       #MyWord := "EPICSToPLC"."Word"[#EPICSToPLCDataBlockOffset + 0];
       "EPICSToPLC"."Word"[#EPICSToPLCDataBlockOffset + 0] := 0;
       #"Cmd_Stop_system" := #MyBoolsinWord[8];    //EPICSName: Cmd_Stop_system
       #"Cmd_Start_system" := #MyBoolsinWord[9];    //EPICSName: Cmd_Start_system
       #"Cmd_Stand_by_4K" := #MyBoolsinWord[10];    //EPICSName: Cmd_Stand_by_4K
       #"Cmd_Stand_by_2K" := #MyBoolsinWord[11];    //EPICSName: Cmd_Stand_by_2K
       #"Cmd_Nominal_2K_RF" := #MyBoolsinWord[12];    //EPICSName: Cmd_Nominal_2K_RF
       #"Cmd_Stand_by_300K" := #MyBoolsinWord[13];    //EPICSName: Cmd_Stand_by_300K
       #"Cmd_Stand_by_80K" := #MyBoolsinWord[14];    //EPICSName: Cmd_Stand_by_80K
       #"Cmd_Reset" := #MyBoolsinWord[15];    //EPICSName: Cmd_Reset
    Else
       #DEVICE_PARAM_OK := FALSE; //Invalid Hash
    END_IF;
END_FUNCTION_BLOCK
FUNCTION_BLOCK "DEVTYPE_C3S_PID"
{ S7_Optimized_Access := 'TRUE' }
VERSION : 1.0
   VAR_INPUT
      "OpMode_Auto" { ExternalAccessible := 'True'; ExternalVisible := 'False'; ExternalWritable := 'False'; } : BOOL;   //EPICS Status variable: OpMode_Auto
      "OpMode_Manual" { ExternalAccessible := 'True'; ExternalVisible := 'False'; ExternalWritable := 'False'; } : BOOL;   //EPICS Status variable: OpMode_Manual
      "OpMode_Forced" { ExternalAccessible := 'True'; ExternalVisible := 'False'; ExternalWritable := 'False'; } : BOOL;   //EPICS Status variable: OpMode_Forced
      "PID_Color" { ExternalAccessible := 'True'; ExternalVisible := 'False'; ExternalWritable := 'False'; } : INT;   //EPICS Status variable: PID_Color
      "LMN" { ExternalAccessible := 'True'; ExternalVisible := 'False'; ExternalWritable := 'False'; } : REAL;   //EPICS Status variable: LMN
      "LMN_P" { ExternalAccessible := 'True'; ExternalVisible := 'False'; ExternalWritable := 'False'; } : REAL;   //EPICS Status variable: LMN_P
      "LMN_I" { ExternalAccessible := 'True'; ExternalVisible := 'False'; ExternalWritable := 'False'; } : REAL;   //EPICS Status variable: LMN_I
      "LMN_D" { ExternalAccessible := 'True'; ExternalVisible := 'False'; ExternalWritable := 'False'; } : REAL;   //EPICS Status variable: LMN_D
      "PID_DIF" { ExternalAccessible := 'True'; ExternalVisible := 'False'; ExternalWritable := 'False'; } : REAL;   //EPICS Status variable: PID_DIF
      "PV" { ExternalAccessible := 'True'; ExternalVisible := 'False'; ExternalWritable := 'False'; } : REAL;   //EPICS Status variable: PV
      "MAN_SP" { ExternalAccessible := 'True'; ExternalVisible := 'False'; ExternalWritable := 'False'; } : REAL;   //EPICS Status variable: MAN_SP
      "PID_Cycle" { ExternalAccessible := 'True'; ExternalVisible := 'False'; ExternalWritable := 'False'; } : INT;   //EPICS Status variable: PID_Cycle
      "ProcValueName" { ExternalAccessible := 'True'; ExternalVisible := 'False'; ExternalWritable := 'False'; } : STRING;   //EPICS Status variable: ProcValueName
      "ProcValueEGU" { ExternalAccessible := 'True'; ExternalVisible := 'False'; ExternalWritable := 'False'; } : STRING;   //EPICS Status variable: ProcValueEGU
      "Inhibit_Manual" { ExternalAccessible := 'True'; ExternalVisible := 'False'; ExternalWritable := 'False'; } : BOOL;   //EPICS Status variable: Inhibit_Manual
      "Inhibit_Force" { ExternalAccessible := 'True'; ExternalVisible := 'False'; ExternalWritable := 'False'; } : BOOL;   //EPICS Status variable: Inhibit_Force
      "Inhibit_Lock" { ExternalAccessible := 'True'; ExternalVisible := 'False'; ExternalWritable := 'False'; } : BOOL;   //EPICS Status variable: Inhibit_Lock
      "MoveInterlock" { ExternalAccessible := 'True'; ExternalVisible := 'False'; ExternalWritable := 'False'; } : BOOL;   //EPICS Status variable: MoveInterlock
      "GroupInterlock" { ExternalAccessible := 'True'; ExternalVisible := 'False'; ExternalWritable := 'False'; } : BOOL;   //EPICS Status variable: GroupInterlock
      "EnableAutoBtn" { ExternalAccessible := 'True'; ExternalVisible := 'False'; ExternalWritable := 'False'; } : BOOL;   //EPICS Status variable: EnableAutoBtn
      "EnableManualBtn" { ExternalAccessible := 'True'; ExternalVisible := 'False'; ExternalWritable := 'False'; } : BOOL;   //EPICS Status variable: EnableManualBtn
      "EnableForcedBtn" { ExternalAccessible := 'True'; ExternalVisible := 'False'; ExternalWritable := 'False'; } : BOOL;   //EPICS Status variable: EnableForcedBtn
      "EnablePIDConf" { ExternalAccessible := 'True'; ExternalVisible := 'False'; ExternalWritable := 'False'; } : BOOL;   //EPICS Status variable: EnablePIDConf
      "LatchAlarm" { ExternalAccessible := 'True'; ExternalVisible := 'False'; ExternalWritable := 'False'; } : BOOL;   //EPICS Status variable: LatchAlarm
      "GroupAlarm" { ExternalAccessible := 'True'; ExternalVisible := 'False'; ExternalWritable := 'False'; } : BOOL;   //EPICS Status variable: GroupAlarm
      "EnableBlkCtrl" { ExternalAccessible := 'True'; ExternalVisible := 'False'; ExternalWritable := 'False'; } : BOOL;   //EPICS Status variable: EnableBlkCtrl
      "EnableForceValBtn" { ExternalAccessible := 'True'; ExternalVisible := 'False'; ExternalWritable := 'False'; } : BOOL;   //EPICS Status variable: EnableForceValBtn
      "DevLocked" { ExternalAccessible := 'True'; ExternalVisible := 'False'; ExternalWritable := 'False'; } : BOOL;   //EPICS Status variable: DevLocked
      "Faceplate_LockID" { ExternalAccessible := 'True'; ExternalVisible := 'False'; ExternalWritable := 'False'; } : DINT;   //EPICS Status variable: Faceplate_LockID
      "BlockIcon_LockID" { ExternalAccessible := 'True'; ExternalVisible := 'False'; ExternalWritable := 'False'; } : DINT;   //EPICS Status variable: BlockIcon_LockID
      "LMN_HLIM" { ExternalAccessible := 'True'; ExternalVisible := 'False'; ExternalWritable := 'False'; } : BOOL;   //EPICS Status variable: LMN_HLIM
      "LMN_LLIM" { ExternalAccessible := 'True'; ExternalVisible := 'False'; ExternalWritable := 'False'; } : BOOL;   //EPICS Status variable: LMN_LLIM
      "IO_Error" { ExternalAccessible := 'True'; ExternalVisible := 'False'; ExternalWritable := 'False'; } : BOOL;   //EPICS Status variable: IO_Error
      "Input_Module_Error" { ExternalAccessible := 'True'; ExternalVisible := 'False'; ExternalWritable := 'False'; } : BOOL;   //EPICS Status variable: Input_Module_Error
      "Output_Module_Error" { ExternalAccessible := 'True'; ExternalVisible := 'False'; ExternalWritable := 'False'; } : BOOL;   //EPICS Status variable: Output_Module_Error
      "Discrepancy_Error" { ExternalAccessible := 'True'; ExternalVisible := 'False'; ExternalWritable := 'False'; } : BOOL;   //EPICS Status variable: Discrepancy_Error
      "ContDeviceInMan" { ExternalAccessible := 'True'; ExternalVisible := 'False'; ExternalWritable := 'False'; } : BOOL;   //EPICS Status variable: ContDeviceInMan
      "FB_Gain" { ExternalAccessible := 'True'; ExternalVisible := 'False'; ExternalWritable := 'False'; } : REAL;   //EPICS Status variable: FB_Gain
      "FB_TI" { ExternalAccessible := 'True'; ExternalVisible := 'False'; ExternalWritable := 'False'; } : DINT;   //EPICS Status variable: FB_TI
      "FB_TD" { ExternalAccessible := 'True'; ExternalVisible := 'False'; ExternalWritable := 'False'; } : DINT;   //EPICS Status variable: FB_TD
      "FB_DEADB" { ExternalAccessible := 'True'; ExternalVisible := 'False'; ExternalWritable := 'False'; } : REAL;   //EPICS Status variable: FB_DEADB
      "FB_LMN_HLIM" { ExternalAccessible := 'True'; ExternalVisible := 'False'; ExternalWritable := 'False'; } : REAL;   //EPICS Status variable: FB_LMN_HLIM
      "FB_LMN_LLIM" { ExternalAccessible := 'True'; ExternalVisible := 'False'; ExternalWritable := 'False'; } : REAL;   //EPICS Status variable: FB_LMN_LLIM
      "FB_ForcePosition" { ExternalAccessible := 'True'; ExternalVisible := 'False'; ExternalWritable := 'False'; } : REAL;   //EPICS Status variable: FB_ForcePosition
      "FB_Setpoint" { ExternalAccessible := 'True'; ExternalVisible := 'False'; ExternalWritable := 'False'; } : REAL;   //EPICS Status variable: FB_Setpoint
      "FB_Step" { ExternalAccessible := 'True'; ExternalVisible := 'False'; ExternalWritable := 'False'; } : REAL;   //EPICS Status variable: FB_Step
      "FB_Manipulated" { ExternalAccessible := 'True'; ExternalVisible := 'False'; ExternalWritable := 'False'; } : REAL;   //EPICS Status variable: FB_Manipulated
      "FB_P_ActionState" { ExternalAccessible := 'True'; ExternalVisible := 'False'; ExternalWritable := 'False'; } : BOOL;   //EPICS Status variable: FB_P_ActionState
      "FB_I_ActionState" { ExternalAccessible := 'True'; ExternalVisible := 'False'; ExternalWritable := 'False'; } : BOOL;   //EPICS Status variable: FB_I_ActionState
      "FB_D_ActionState" { ExternalAccessible := 'True'; ExternalVisible := 'False'; ExternalWritable := 'False'; } : BOOL;   //EPICS Status variable: FB_D_ActionState
      "FB_SS_State" { ExternalAccessible := 'True'; ExternalVisible := 'False'; ExternalWritable := 'False'; } : BOOL;   //EPICS Status variable: FB_SS_State
      "FB_SS_Value" { ExternalAccessible := 'True'; ExternalVisible := 'False'; ExternalWritable := 'False'; } : REAL;   //EPICS Status variable: FB_SS_Value
      "MeasValue_Msg" { ExternalAccessible := 'True'; ExternalVisible := 'False'; ExternalWritable := 'False'; } : STRING;   //EPICS Status variable: Measured_Value_Msg
   EPICSToPLCLength { ExternalAccessible := 'False'; ExternalVisible := 'False'; ExternalWritable := 'False'; } : Int;   // Length of device command register array (in words)
   EPICSToPLCDataBlockOffset { ExternalAccessible := 'False'; ExternalVisible := 'False'; ExternalWritable := 'False'; } : Int;   // Offset in EPICS->PLC comms block where this device data resides (in words)
   PLCToEPICSLength { ExternalAccessible := 'False'; ExternalVisible := 'False'; ExternalWritable := 'False'; } : Int;   // Length of device status register array (in words)
   PLCToEPICSDataBlockOffset { ExternalAccessible := 'False'; ExternalVisible := 'False'; ExternalWritable := 'False'; } : Int;   // Offset in PLC->EPICS comms block where this device data resides (in words)
   END_VAR
   VAR_OUTPUT
      "Cmd_Auto" { ExternalAccessible := 'True'; ExternalVisible := 'False'; ExternalWritable := 'False'; } : BOOL;   //EPICS Command variable: Cmd_Auto
      "Cmd_Manual" { ExternalAccessible := 'True'; ExternalVisible := 'False'; ExternalWritable := 'False'; } : BOOL;   //EPICS Command variable: Cmd_Manual
      "Cmd_Force" { ExternalAccessible := 'True'; ExternalVisible := 'False'; ExternalWritable := 'False'; } : BOOL;   //EPICS Command variable: Cmd_Force
      "Cmd_EnablePID_Conf" { ExternalAccessible := 'True'; ExternalVisible := 'False'; ExternalWritable := 'False'; } : BOOL;   //EPICS Command variable: Cmd_EnablePID_Conf
      "Cmd_DisablePID_Conf" { ExternalAccessible := 'True'; ExternalVisible := 'False'; ExternalWritable := 'False'; } : BOOL;   //EPICS Command variable: Cmd_DisablePID_Conf
      "Cmd_P_ON" { ExternalAccessible := 'True'; ExternalVisible := 'False'; ExternalWritable := 'False'; } : BOOL;   //EPICS Command variable: Cmd_P_ON
      "Cmd_P_OFF" { ExternalAccessible := 'True'; ExternalVisible := 'False'; ExternalWritable := 'False'; } : BOOL;   //EPICS Command variable: Cmd_P_OFF
      "Cmd_I_ON" { ExternalAccessible := 'True'; ExternalVisible := 'False'; ExternalWritable := 'False'; } : BOOL;   //EPICS Command variable: Cmd_I_ON
      "Cmd_I_OFF" { ExternalAccessible := 'True'; ExternalVisible := 'False'; ExternalWritable := 'False'; } : BOOL;   //EPICS Command variable: Cmd_I_OFF
      "Cmd_D_ON" { ExternalAccessible := 'True'; ExternalVisible := 'False'; ExternalWritable := 'False'; } : BOOL;   //EPICS Command variable: Cmd_D_ON
      "Cmd_D_OFF" { ExternalAccessible := 'True'; ExternalVisible := 'False'; ExternalWritable := 'False'; } : BOOL;   //EPICS Command variable: Cmd_D_OFF
      "Cmd_AckAlarm" { ExternalAccessible := 'True'; ExternalVisible := 'False'; ExternalWritable := 'False'; } : BOOL;   //EPICS Command variable: Cmd_AckAlarm
      "Cmd_ForceValInp" { ExternalAccessible := 'True'; ExternalVisible := 'False'; ExternalWritable := 'False'; } : BOOL;   //EPICS Command variable: Cmd_ForceValInp
      "Cmd_ForceValOut" { ExternalAccessible := 'True'; ExternalVisible := 'False'; ExternalWritable := 'False'; } : BOOL;   //EPICS Command variable: Cmd_ForceValOut
      "Cmd_ForceUnlock" { ExternalAccessible := 'True'; ExternalVisible := 'False'; ExternalWritable := 'False'; } : BOOL;   //EPICS Command variable: Cmd_ForceUnlock
      "Cmd_DevLock" { ExternalAccessible := 'True'; ExternalVisible := 'False'; ExternalWritable := 'False'; } : BOOL;   //EPICS Command variable: Cmd_DevLock
      "Cmd_DevUnlock" { ExternalAccessible := 'True'; ExternalVisible := 'False'; ExternalWritable := 'False'; } : BOOL;   //EPICS Command variable: Cmd_DevUnlock
      "P_Gain" { ExternalAccessible := 'True'; ExternalVisible := 'False'; ExternalWritable := 'False'; } : REAL;   //EPICS Parameter variable: P_Gain
      "P_TI" { ExternalAccessible := 'True'; ExternalVisible := 'False'; ExternalWritable := 'False'; } : DINT;   //EPICS Parameter variable: P_TI
      "P_TD" { ExternalAccessible := 'True'; ExternalVisible := 'False'; ExternalWritable := 'False'; } : DINT;   //EPICS Parameter variable: P_TD
      "P_DEADB" { ExternalAccessible := 'True'; ExternalVisible := 'False'; ExternalWritable := 'False'; } : REAL;   //EPICS Parameter variable: P_DEADB
      "P_LMN_HLIM" { ExternalAccessible := 'True'; ExternalVisible := 'False'; ExternalWritable := 'False'; } : REAL;   //EPICS Parameter variable: P_LMN_HLIM
      "P_LMN_LLIM" { ExternalAccessible := 'True'; ExternalVisible := 'False'; ExternalWritable := 'False'; } : REAL;   //EPICS Parameter variable: P_LMN_LLIM
      "P_ForcePosition" { ExternalAccessible := 'True'; ExternalVisible := 'False'; ExternalWritable := 'False'; } : REAL;   //EPICS Parameter variable: P_ForcePosition
      "P_Setpoint" { ExternalAccessible := 'True'; ExternalVisible := 'False'; ExternalWritable := 'False'; } : REAL;   //EPICS Parameter variable: P_Setpoint
      "P_Manipulated" { ExternalAccessible := 'True'; ExternalVisible := 'False'; ExternalWritable := 'False'; } : REAL;   //EPICS Parameter variable: P_Manipulated
      "P_Step" { ExternalAccessible := 'True'; ExternalVisible := 'False'; ExternalWritable := 'False'; } : REAL;   //EPICS Parameter variable: P_Step
      "P_Faceplate_LockID" { ExternalAccessible := 'True'; ExternalVisible := 'False'; ExternalWritable := 'False'; } : DINT;   //EPICS Parameter variable: P_Faceplate_LockID
      "P_BlockIcon_LockID" { ExternalAccessible := 'True'; ExternalVisible := 'False'; ExternalWritable := 'False'; } : DINT;   //EPICS Parameter variable: P_BlockIcon_LockID
      DEVICE_PARAM_OK { ExternalAccessible := 'False'; ExternalVisible := 'False'; ExternalWritable := 'False'; } : Bool;
   END_VAR
   VAR_IN_OUT
   END_VAR
   Var DB_SPECIFIC
      MyWord { ExternalAccessible := 'False'; ExternalVisible := 'False'; ExternalWritable := 'False'; } : Word;
      MyBytesinWord { ExternalAccessible := 'False'; ExternalVisible := 'False'; ExternalWritable := 'False'; } AT MyWord : Array[0..1] of Byte;
      MyBoolsinWord { ExternalAccessible := 'False'; ExternalVisible := 'False'; ExternalWritable := 'False'; } AT MyWord : Array[0..15] of Bool;
      MyDInt { ExternalAccessible := 'False'; ExternalVisible := 'False'; ExternalWritable := 'False'; } : DInt;
      MyWordsinDint { ExternalAccessible := 'False'; ExternalVisible := 'False'; ExternalWritable := 'False'; } AT MyDInt : Array[0..1] of Word;
      MyReal { ExternalAccessible := 'False'; ExternalVisible := 'False'; ExternalWritable := 'False'; } : Real;
      MyWordsinReal { ExternalAccessible := 'False'; ExternalVisible := 'False'; ExternalWritable := 'False'; } AT MyReal : Array[0..1] of Word;
      MyInt { ExternalAccessible := 'False'; ExternalVisible := 'False'; ExternalWritable := 'False'; } : Int;
      MyWordinInt { ExternalAccessible := 'False'; ExternalVisible := 'False'; ExternalWritable := 'False'; } AT MyInt : Word;
      MyDWord { ExternalAccessible := 'False'; ExternalVisible := 'False'; ExternalWritable := 'False'; } : DWord;
      MyWordsinDWord { ExternalAccessible := 'False'; ExternalVisible := 'False'; ExternalWritable := 'False'; } AT MyDWord : Array[0..1] of Word;
      MyTime { ExternalAccessible := 'False'; ExternalVisible := 'False'; ExternalWritable := 'False'; } : Time;
      MyWordsinTime { ExternalAccessible := 'False'; ExternalVisible := 'False'; ExternalWritable := 'False'; } AT MyTime : Array[0..1] of Word;
      MyString { ExternalAccessible := 'False'; ExternalVisible := 'False'; ExternalWritable := 'False'; } : String[40];
      MyWordsinString { ExternalAccessible := 'False'; ExternalVisible := 'False'; ExternalWritable := 'False'; } AT MyString : Array[0..20] of Word;
   END_VAR
   VAR_TEMP
      HashModbus : DInt;
      HashIFA : DInt;
      HashTIAMap : DInt;
      i : Int;
   END_VAR
    //Author: Miklos Boros (miklos.boros@esss.se), Copyrigth 2017-2020 by European Spallation Source, Lund
    //This block was generated by PLCFactory, please don't change it MANUALLY!
    //Input File Name: Spk-000CDL_Cryo-PLC-010-template-IFA-20220922093722.ifa
    //Generated: 20220922093722
    //According to HASH: 457744924
    //Device type: C3S_PID
    //Description: This function does the variable mapping for a device. All device-variable will be linked to an interface variable defined in this block.

    //********************************************
    //****************HASH check******************
    //********************************************


    #MyWordsinDint[0] := "EPICSToPLC"."Word"[0];
    #MyWordsinDint[1] := "EPICSToPLC"."Word"[1];
    #HashModbus := #MyDInt; //Hash from EPICS/ModbusTCP

    #HashIFA := 457744924; //Hash from Interface Factory as a constant

    #MyWordsinDint[0] := "PLCToEPICS"."Word"[0];
    #MyWordsinDint[1] := "PLCToEPICS"."Word"[1];
    #HashTIAMap := #MyDInt; //Hash from PLCFactory TIA Map


    IF ((#HashIFA = #HashModbus) AND (#HashModbus = #HashTIAMap)) THEN //Check CRCs
        #DEVICE_PARAM_OK := TRUE;
       //##################################### ICS HWI ###############################################
       //############################  ICS Instrument Library     ####################################
       //#  PLC Sample Code in VersionDog: ICS_LIBRARY_MASTER_PLC                                   ##
       //#  CCDB device types: ICS_xxxxx                                                            ##
       //#  EPICS HMI (Block Icons/Faceplates)@ GitLab. Projekt: Cryo / CryogenicsLibrary / CryoLib ##
       //#                                                                                          ##
       //#                                 PID - PID Control                                        ##
       //#                                                                                          ##
       //#                                                                                          ##
       //###########################           Version: 1.2           ################################
       //Author:	Zoltan Madi
       //Date:		13-12-2019
       //Version:  v1.2
       //Changes:  Added "MeasValue_Msg"
       //###########################           Version: 1.1           ################################
       //Author:	Johannes Kazantzidis
       //Date:		13-12-2019
       //Version:  v1.1
       //Changes:  Added alarm signal "Discrepancy_Error"
       //###########################           Version: 1.0           ################################
       //Author:	Miklos Boros
       //Date:		01-09-2019
       //Version:  v1.0
       //Changes:  First release and alarm signal "Discrepancy_Error"
       //#############################################################################################
       //###########################
       //STATUS BLOCK
       //###########################
       //Operation modes
       //OPI buttons
       //PID

    //********************************************
    //*************STATUS VARIABLES***************
    //********************************************


       #MyWord := W#0;
       #MyBoolsinWord[8] := #"OpMode_Auto";    //EPICSName: OpMode_Auto
       #MyBoolsinWord[9] := #"OpMode_Manual";    //EPICSName: OpMode_Manual
       #MyBoolsinWord[10] := #"OpMode_Forced";    //EPICSName: OpMode_Forced
       "PLCToEPICS"."Word"[#PLCToEPICSDataBlockOffset + 0] := #MyWord;

       #MyInt := #"PID_Color";    //EPICSName: PID_Color
       "PLCToEPICS"."Word"[#PLCToEPICSDataBlockOffset + 1] := #MyWordinInt;

       #MyReal := #"LMN";    //EPICSName: LMN
       "PLCToEPICS"."Word"[#PLCToEPICSDataBlockOffset + 2] := #MyWordsinReal[0];
       "PLCToEPICS"."Word"[#PLCToEPICSDataBlockOffset + 3] := #MyWordsinReal[1];

       #MyReal := #"LMN_P";    //EPICSName: LMN_P
       "PLCToEPICS"."Word"[#PLCToEPICSDataBlockOffset + 4] := #MyWordsinReal[0];
       "PLCToEPICS"."Word"[#PLCToEPICSDataBlockOffset + 5] := #MyWordsinReal[1];

       #MyReal := #"LMN_I";    //EPICSName: LMN_I
       "PLCToEPICS"."Word"[#PLCToEPICSDataBlockOffset + 6] := #MyWordsinReal[0];
       "PLCToEPICS"."Word"[#PLCToEPICSDataBlockOffset + 7] := #MyWordsinReal[1];

       #MyReal := #"LMN_D";    //EPICSName: LMN_D
       "PLCToEPICS"."Word"[#PLCToEPICSDataBlockOffset + 8] := #MyWordsinReal[0];
       "PLCToEPICS"."Word"[#PLCToEPICSDataBlockOffset + 9] := #MyWordsinReal[1];

       #MyReal := #"PID_DIF";    //EPICSName: PID_DIF
       "PLCToEPICS"."Word"[#PLCToEPICSDataBlockOffset + 10] := #MyWordsinReal[0];
       "PLCToEPICS"."Word"[#PLCToEPICSDataBlockOffset + 11] := #MyWordsinReal[1];

       #MyReal := #"PV";    //EPICSName: PV
       "PLCToEPICS"."Word"[#PLCToEPICSDataBlockOffset + 12] := #MyWordsinReal[0];
       "PLCToEPICS"."Word"[#PLCToEPICSDataBlockOffset + 13] := #MyWordsinReal[1];

       #MyReal := #"MAN_SP";    //EPICSName: MAN_SP
       "PLCToEPICS"."Word"[#PLCToEPICSDataBlockOffset + 14] := #MyWordsinReal[0];
       "PLCToEPICS"."Word"[#PLCToEPICSDataBlockOffset + 15] := #MyWordsinReal[1];

       #MyInt := #"PID_Cycle";    //EPICSName: PID_Cycle
       "PLCToEPICS"."Word"[#PLCToEPICSDataBlockOffset + 16] := #MyWordinInt;

       // Clear the buffer of any residual data, but skip the first word as that is the actual and maximum length
       FOR #i:=1 TO 20 DO
            #MyWordsinString[#i] := 0;
       END_FOR;
       #MyString := #"ProcValueName";  //EPICSName: ProcValueName
       FOR #i:=0 TO 18 DO
            "PLCToEPICS"."Word"[#PLCToEPICSDataBlockOffset + 17 + #i] := #MyWordsinString[#i + 1];
       END_FOR;
       // Terminate C-string
       "PLCToEPICS"."Word"[#PLCToEPICSDataBlockOffset + 17 + 19] := #MyWordsinString[20] & 16#FF00;

       // Clear the buffer of any residual data, but skip the first word as that is the actual and maximum length
       FOR #i:=1 TO 20 DO
            #MyWordsinString[#i] := 0;
       END_FOR;
       #MyString := #"ProcValueEGU";  //EPICSName: ProcValueEGU
       FOR #i:=0 TO 2 DO
            "PLCToEPICS"."Word"[#PLCToEPICSDataBlockOffset + 37 + #i] := #MyWordsinString[#i + 1];
       END_FOR;
       // Terminate C-string
       "PLCToEPICS"."Word"[#PLCToEPICSDataBlockOffset + 37 + 3] := 0;

       #MyWord := W#0;
       #MyBoolsinWord[8] := #"Inhibit_Manual";    //EPICSName: Inhibit_Manual
       #MyBoolsinWord[9] := #"Inhibit_Force";    //EPICSName: Inhibit_Force
       #MyBoolsinWord[10] := #"Inhibit_Lock";    //EPICSName: Inhibit_Lock
       #MyBoolsinWord[11] := #"MoveInterlock";    //EPICSName: MoveInterlock
       #MyBoolsinWord[12] := #"GroupInterlock";    //EPICSName: GroupInterlock
       #MyBoolsinWord[13] := #"EnableAutoBtn";    //EPICSName: EnableAutoBtn
       #MyBoolsinWord[14] := #"EnableManualBtn";    //EPICSName: EnableManualBtn
       #MyBoolsinWord[15] := #"EnableForcedBtn";    //EPICSName: EnableForcedBtn
       #MyBoolsinWord[0] := #"EnablePIDConf";    //EPICSName: EnablePIDConf
       #MyBoolsinWord[1] := #"LatchAlarm";    //EPICSName: LatchAlarm
       #MyBoolsinWord[2] := #"GroupAlarm";    //EPICSName: GroupAlarm
       #MyBoolsinWord[3] := #"EnableBlkCtrl";    //EPICSName: EnableBlkCtrl
       #MyBoolsinWord[4] := #"EnableForceValBtn";    //EPICSName: EnableForceValBtn
       #MyBoolsinWord[5] := #"DevLocked";    //EPICSName: DevLocked
       "PLCToEPICS"."Word"[#PLCToEPICSDataBlockOffset + 41] := #MyWord;

       #MyDInt := #"Faceplate_LockID";    //EPICSName: Faceplate_LockID
       "PLCToEPICS"."Word"[#PLCToEPICSDataBlockOffset + 42] := #MyWordsinDint[0];
       "PLCToEPICS"."Word"[#PLCToEPICSDataBlockOffset + 43] := #MyWordsinDint[1];

       #MyDInt := #"BlockIcon_LockID";    //EPICSName: BlockIcon_LockID
       "PLCToEPICS"."Word"[#PLCToEPICSDataBlockOffset + 44] := #MyWordsinDint[0];
       "PLCToEPICS"."Word"[#PLCToEPICSDataBlockOffset + 45] := #MyWordsinDint[1];

       #MyWord := W#0;
       #MyBoolsinWord[8] := #"LMN_HLIM";    //EPICSName: LMN_HLIM
       #MyBoolsinWord[9] := #"LMN_LLIM";    //EPICSName: LMN_LLIM
       #MyBoolsinWord[10] := #"IO_Error";    //EPICSName: IO_Error
       #MyBoolsinWord[11] := #"Input_Module_Error";    //EPICSName: Input_Module_Error
       #MyBoolsinWord[12] := #"Output_Module_Error";    //EPICSName: Output_Module_Error
       #MyBoolsinWord[13] := #"Discrepancy_Error";    //EPICSName: Discrepancy_Error
       #MyBoolsinWord[14] := #"ContDeviceInMan";    //EPICSName: ContDeviceInMan
       "PLCToEPICS"."Word"[#PLCToEPICSDataBlockOffset + 46] := #MyWord;

       #MyReal := #"FB_Gain";    //EPICSName: FB_Gain
       "PLCToEPICS"."Word"[#PLCToEPICSDataBlockOffset + 47] := #MyWordsinReal[0];
       "PLCToEPICS"."Word"[#PLCToEPICSDataBlockOffset + 48] := #MyWordsinReal[1];

       #MyDInt := #"FB_TI";    //EPICSName: FB_TI
       "PLCToEPICS"."Word"[#PLCToEPICSDataBlockOffset + 49] := #MyWordsinDint[0];
       "PLCToEPICS"."Word"[#PLCToEPICSDataBlockOffset + 50] := #MyWordsinDint[1];

       #MyDInt := #"FB_TD";    //EPICSName: FB_TD
       "PLCToEPICS"."Word"[#PLCToEPICSDataBlockOffset + 51] := #MyWordsinDint[0];
       "PLCToEPICS"."Word"[#PLCToEPICSDataBlockOffset + 52] := #MyWordsinDint[1];

       #MyReal := #"FB_DEADB";    //EPICSName: FB_DEADB
       "PLCToEPICS"."Word"[#PLCToEPICSDataBlockOffset + 53] := #MyWordsinReal[0];
       "PLCToEPICS"."Word"[#PLCToEPICSDataBlockOffset + 54] := #MyWordsinReal[1];

       #MyReal := #"FB_LMN_HLIM";    //EPICSName: FB_LMN_HLIM
       "PLCToEPICS"."Word"[#PLCToEPICSDataBlockOffset + 55] := #MyWordsinReal[0];
       "PLCToEPICS"."Word"[#PLCToEPICSDataBlockOffset + 56] := #MyWordsinReal[1];

       #MyReal := #"FB_LMN_LLIM";    //EPICSName: FB_LMN_LLIM
       "PLCToEPICS"."Word"[#PLCToEPICSDataBlockOffset + 57] := #MyWordsinReal[0];
       "PLCToEPICS"."Word"[#PLCToEPICSDataBlockOffset + 58] := #MyWordsinReal[1];

       #MyReal := #"FB_ForcePosition";    //EPICSName: FB_ForcePosition
       "PLCToEPICS"."Word"[#PLCToEPICSDataBlockOffset + 59] := #MyWordsinReal[0];
       "PLCToEPICS"."Word"[#PLCToEPICSDataBlockOffset + 60] := #MyWordsinReal[1];

       #MyReal := #"FB_Setpoint";    //EPICSName: FB_Setpoint
       "PLCToEPICS"."Word"[#PLCToEPICSDataBlockOffset + 61] := #MyWordsinReal[0];
       "PLCToEPICS"."Word"[#PLCToEPICSDataBlockOffset + 62] := #MyWordsinReal[1];

       #MyReal := #"FB_Step";    //EPICSName: FB_Step
       "PLCToEPICS"."Word"[#PLCToEPICSDataBlockOffset + 63] := #MyWordsinReal[0];
       "PLCToEPICS"."Word"[#PLCToEPICSDataBlockOffset + 64] := #MyWordsinReal[1];

       #MyReal := #"FB_Manipulated";    //EPICSName: FB_Manipulated
       "PLCToEPICS"."Word"[#PLCToEPICSDataBlockOffset + 65] := #MyWordsinReal[0];
       "PLCToEPICS"."Word"[#PLCToEPICSDataBlockOffset + 66] := #MyWordsinReal[1];

       #MyWord := W#0;
       #MyBoolsinWord[8] := #"FB_P_ActionState";    //EPICSName: FB_P_ActionState
       #MyBoolsinWord[9] := #"FB_I_ActionState";    //EPICSName: FB_I_ActionState
       #MyBoolsinWord[10] := #"FB_D_ActionState";    //EPICSName: FB_D_ActionState
       #MyBoolsinWord[11] := #"FB_SS_State";    //EPICSName: FB_SS_State
       "PLCToEPICS"."Word"[#PLCToEPICSDataBlockOffset + 67] := #MyWord;

       #MyReal := #"FB_SS_Value";    //EPICSName: FB_SS_Value
       "PLCToEPICS"."Word"[#PLCToEPICSDataBlockOffset + 68] := #MyWordsinReal[0];
       "PLCToEPICS"."Word"[#PLCToEPICSDataBlockOffset + 69] := #MyWordsinReal[1];

       // Clear the buffer of any residual data, but skip the first word as that is the actual and maximum length
       FOR #i:=1 TO 20 DO
            #MyWordsinString[#i] := 0;
       END_FOR;
       #MyString := #"MeasValue_Msg";  //EPICSName: Measured_Value_Msg
       FOR #i:=0 TO 18 DO
            "PLCToEPICS"."Word"[#PLCToEPICSDataBlockOffset + 70 + #i] := #MyWordsinString[#i + 1];
       END_FOR;
       // Terminate C-string
       "PLCToEPICS"."Word"[#PLCToEPICSDataBlockOffset + 70 + 19] := #MyWordsinString[20] & 16#FF00;

    //********************************************
    //*************COMMAND VARIABLES**************
    //********************************************


       #MyWord := "EPICSToPLC"."Word"[#EPICSToPLCDataBlockOffset + 0];
       "EPICSToPLC"."Word"[#EPICSToPLCDataBlockOffset + 0] := 0;
       #"Cmd_Auto" := #MyBoolsinWord[8];    //EPICSName: Cmd_Auto
       #"Cmd_Manual" := #MyBoolsinWord[9];    //EPICSName: Cmd_Manual
       #"Cmd_Force" := #MyBoolsinWord[10];    //EPICSName: Cmd_Force
       #"Cmd_EnablePID_Conf" := #MyBoolsinWord[11];    //EPICSName: Cmd_EnablePID_Conf
       #"Cmd_DisablePID_Conf" := #MyBoolsinWord[12];    //EPICSName: Cmd_DisablePID_Conf
       #"Cmd_P_ON" := #MyBoolsinWord[13];    //EPICSName: Cmd_P_ON
       #"Cmd_P_OFF" := #MyBoolsinWord[14];    //EPICSName: Cmd_P_OFF
       #"Cmd_I_ON" := #MyBoolsinWord[15];    //EPICSName: Cmd_I_ON
       #"Cmd_I_OFF" := #MyBoolsinWord[0];    //EPICSName: Cmd_I_OFF
       #"Cmd_D_ON" := #MyBoolsinWord[1];    //EPICSName: Cmd_D_ON
       #"Cmd_D_OFF" := #MyBoolsinWord[2];    //EPICSName: Cmd_D_OFF
       #"Cmd_AckAlarm" := #MyBoolsinWord[3];    //EPICSName: Cmd_AckAlarm
       #"Cmd_ForceValInp" := #MyBoolsinWord[4];    //EPICSName: Cmd_ForceValInp
       #"Cmd_ForceValOut" := #MyBoolsinWord[5];    //EPICSName: Cmd_ForceValOut
       #"Cmd_ForceUnlock" := #MyBoolsinWord[6];    //EPICSName: Cmd_ForceUnlock
       #"Cmd_DevLock" := #MyBoolsinWord[7];    //EPICSName: Cmd_DevLock

       #MyWord := "EPICSToPLC"."Word"[#EPICSToPLCDataBlockOffset + 1];
       "EPICSToPLC"."Word"[#EPICSToPLCDataBlockOffset + 1] := 0;
       #"Cmd_DevUnlock" := #MyBoolsinWord[8];    //EPICSName: Cmd_DevUnlock

    //********************************************
    //************PARAMETER VARIABLES*************
    //********************************************


       #MyReal	:= 0.0;
       #MyWordsinReal[0]	:= "EPICSToPLC"."Word"[#EPICSToPLCDataBlockOffset + 2];
       #MyWordsinReal[1]	:= "EPICSToPLC"."Word"[#EPICSToPLCDataBlockOffset + 3];
       #"P_Gain" := #MyReal;    //EPICSName: P_Gain

       #MyDInt	:= 0;
       #MyWordsinDint[0]	:= "EPICSToPLC"."Word"[#EPICSToPLCDataBlockOffset + 4];
       #MyWordsinDint[1]	:= "EPICSToPLC"."Word"[#EPICSToPLCDataBlockOffset + 5];
       #"P_TI" := #MyDInt;    //EPICSName: P_TI

       #MyDInt	:= 0;
       #MyWordsinDint[0]	:= "EPICSToPLC"."Word"[#EPICSToPLCDataBlockOffset + 6];
       #MyWordsinDint[1]	:= "EPICSToPLC"."Word"[#EPICSToPLCDataBlockOffset + 7];
       #"P_TD" := #MyDInt;    //EPICSName: P_TD

       #MyReal	:= 0.0;
       #MyWordsinReal[0]	:= "EPICSToPLC"."Word"[#EPICSToPLCDataBlockOffset + 8];
       #MyWordsinReal[1]	:= "EPICSToPLC"."Word"[#EPICSToPLCDataBlockOffset + 9];
       #"P_DEADB" := #MyReal;    //EPICSName: P_DEADB

       #MyReal	:= 0.0;
       #MyWordsinReal[0]	:= "EPICSToPLC"."Word"[#EPICSToPLCDataBlockOffset + 10];
       #MyWordsinReal[1]	:= "EPICSToPLC"."Word"[#EPICSToPLCDataBlockOffset + 11];
       #"P_LMN_HLIM" := #MyReal;    //EPICSName: P_LMN_HLIM

       #MyReal	:= 0.0;
       #MyWordsinReal[0]	:= "EPICSToPLC"."Word"[#EPICSToPLCDataBlockOffset + 12];
       #MyWordsinReal[1]	:= "EPICSToPLC"."Word"[#EPICSToPLCDataBlockOffset + 13];
       #"P_LMN_LLIM" := #MyReal;    //EPICSName: P_LMN_LLIM

       #MyReal	:= 0.0;
       #MyWordsinReal[0]	:= "EPICSToPLC"."Word"[#EPICSToPLCDataBlockOffset + 14];
       #MyWordsinReal[1]	:= "EPICSToPLC"."Word"[#EPICSToPLCDataBlockOffset + 15];
       #"P_ForcePosition" := #MyReal;    //EPICSName: P_ForcePosition

       #MyReal	:= 0.0;
       #MyWordsinReal[0]	:= "EPICSToPLC"."Word"[#EPICSToPLCDataBlockOffset + 16];
       #MyWordsinReal[1]	:= "EPICSToPLC"."Word"[#EPICSToPLCDataBlockOffset + 17];
       #"P_Setpoint" := #MyReal;    //EPICSName: P_Setpoint

       #MyReal	:= 0.0;
       #MyWordsinReal[0]	:= "EPICSToPLC"."Word"[#EPICSToPLCDataBlockOffset + 18];
       #MyWordsinReal[1]	:= "EPICSToPLC"."Word"[#EPICSToPLCDataBlockOffset + 19];
       #"P_Manipulated" := #MyReal;    //EPICSName: P_Manipulated

       #MyReal	:= 0.0;
       #MyWordsinReal[0]	:= "EPICSToPLC"."Word"[#EPICSToPLCDataBlockOffset + 20];
       #MyWordsinReal[1]	:= "EPICSToPLC"."Word"[#EPICSToPLCDataBlockOffset + 21];
       #"P_Step" := #MyReal;    //EPICSName: P_Step

       #MyDInt	:= 0;
       #MyWordsinDint[0]	:= "EPICSToPLC"."Word"[#EPICSToPLCDataBlockOffset + 22];
       #MyWordsinDint[1]	:= "EPICSToPLC"."Word"[#EPICSToPLCDataBlockOffset + 23];
       #"P_Faceplate_LockID" := #MyDInt;    //EPICSName: P_Faceplate_LockID

       #MyDInt	:= 0;
       #MyWordsinDint[0]	:= "EPICSToPLC"."Word"[#EPICSToPLCDataBlockOffset + 24];
       #MyWordsinDint[1]	:= "EPICSToPLC"."Word"[#EPICSToPLCDataBlockOffset + 25];
       #"P_BlockIcon_LockID" := #MyDInt;    //EPICSName: P_BlockIcon_LockID
    Else
       #DEVICE_PARAM_OK := FALSE; //Invalid Hash
    END_IF;
END_FUNCTION_BLOCK
FUNCTION_BLOCK "DEVTYPE_ICS_CV_PB_SIPART"
{ S7_Optimized_Access := 'TRUE' }
VERSION : 1.0
   VAR_INPUT
      "OpMode_Auto" { ExternalAccessible := 'True'; ExternalVisible := 'False'; ExternalWritable := 'False'; } : BOOL;   //EPICS Status variable: OpMode_Auto
      "OpMode_Manual" { ExternalAccessible := 'True'; ExternalVisible := 'False'; ExternalWritable := 'False'; } : BOOL;   //EPICS Status variable: OpMode_Manual
      "OpMode_Forced" { ExternalAccessible := 'True'; ExternalVisible := 'False'; ExternalWritable := 'False'; } : BOOL;   //EPICS Status variable: OpMode_Forced
      "ValveColor" { ExternalAccessible := 'True'; ExternalVisible := 'False'; ExternalWritable := 'False'; } : INT;   //EPICS Status variable: ValveColor
      "ValvePosition" { ExternalAccessible := 'True'; ExternalVisible := 'False'; ExternalWritable := 'False'; } : REAL;   //EPICS Status variable: ValvePosition
      "ValveSP" { ExternalAccessible := 'True'; ExternalVisible := 'False'; ExternalWritable := 'False'; } : REAL;   //EPICS Status variable: ValveSP
      "ValveMV" { ExternalAccessible := 'True'; ExternalVisible := 'False'; ExternalWritable := 'False'; } : REAL;   //EPICS Status variable: ValveMV
      "Opening" { ExternalAccessible := 'True'; ExternalVisible := 'False'; ExternalWritable := 'False'; } : BOOL;   //EPICS Status variable: Opening
      "Closing" { ExternalAccessible := 'True'; ExternalVisible := 'False'; ExternalWritable := 'False'; } : BOOL;   //EPICS Status variable: Closing
      "StatusRB" { ExternalAccessible := 'True'; ExternalVisible := 'False'; ExternalWritable := 'False'; } : BYTE;   //EPICS Status variable: StatusRB
      "DiscretePosition" { ExternalAccessible := 'True'; ExternalVisible := 'False'; ExternalWritable := 'False'; } : INT;   //EPICS Status variable: DiscretePosition
      "DiscreteStatus" { ExternalAccessible := 'True'; ExternalVisible := 'False'; ExternalWritable := 'False'; } : BYTE;   //EPICS Status variable: DiscreteStatus
      "DiagnosticsCB01" { ExternalAccessible := 'True'; ExternalVisible := 'False'; ExternalWritable := 'False'; } : BYTE;   //EPICS Status variable: DiagnosticsCB01
      "DiagnosticsCB02" { ExternalAccessible := 'True'; ExternalVisible := 'False'; ExternalWritable := 'False'; } : BYTE;   //EPICS Status variable: DiagnosticsCB02
      "DiagnosticsCB03" { ExternalAccessible := 'True'; ExternalVisible := 'False'; ExternalWritable := 'False'; } : BYTE;   //EPICS Status variable: DiagnosticsCB03
      "Inhibit_Manual" { ExternalAccessible := 'True'; ExternalVisible := 'False'; ExternalWritable := 'False'; } : BOOL;   //EPICS Status variable: Inhibit_Manual
      "Inhibit_Force" { ExternalAccessible := 'True'; ExternalVisible := 'False'; ExternalWritable := 'False'; } : BOOL;   //EPICS Status variable: Inhibit_Force
      "Inhibit_Lock" { ExternalAccessible := 'True'; ExternalVisible := 'False'; ExternalWritable := 'False'; } : BOOL;   //EPICS Status variable: Inhibit_Lock
      "GroupInterlock" { ExternalAccessible := 'True'; ExternalVisible := 'False'; ExternalWritable := 'False'; } : BOOL;   //EPICS Status variable: GroupInterlock
      "InterlockMsg" { ExternalAccessible := 'True'; ExternalVisible := 'False'; ExternalWritable := 'False'; } : STRING;   //EPICS Status variable: InterlockMsg
      "MoveInterlock" { ExternalAccessible := 'True'; ExternalVisible := 'False'; ExternalWritable := 'False'; } : BOOL;   //EPICS Status variable: MoveInterlock
      "EnableAutoBtn" { ExternalAccessible := 'True'; ExternalVisible := 'False'; ExternalWritable := 'False'; } : BOOL;   //EPICS Status variable: EnableAutoBtn
      "EnableManualBtn" { ExternalAccessible := 'True'; ExternalVisible := 'False'; ExternalWritable := 'False'; } : BOOL;   //EPICS Status variable: EnableManualBtn
      "EnableForcedBtn" { ExternalAccessible := 'True'; ExternalVisible := 'False'; ExternalWritable := 'False'; } : BOOL;   //EPICS Status variable: EnableForcedBtn
      "EnableBlkCtrl" { ExternalAccessible := 'True'; ExternalVisible := 'False'; ExternalWritable := 'False'; } : BOOL;   //EPICS Status variable: EnableBlkCtrl
      "EnableForceValBtn" { ExternalAccessible := 'True'; ExternalVisible := 'False'; ExternalWritable := 'False'; } : BOOL;   //EPICS Status variable: EnableForceValBtn
      "DevLocked" { ExternalAccessible := 'True'; ExternalVisible := 'False'; ExternalWritable := 'False'; } : BOOL;   //EPICS Status variable: DevLocked
      "Faceplate_LockID" { ExternalAccessible := 'True'; ExternalVisible := 'False'; ExternalWritable := 'False'; } : DINT;   //EPICS Status variable: Faceplate_LockID
      "BlockIcon_LockID" { ExternalAccessible := 'True'; ExternalVisible := 'False'; ExternalWritable := 'False'; } : DINT;   //EPICS Status variable: BlockIcon_LockID
      "LatchAlarm" { ExternalAccessible := 'True'; ExternalVisible := 'False'; ExternalWritable := 'False'; } : BOOL;   //EPICS Status variable: LatchAlarm
      "GroupAlarm" { ExternalAccessible := 'True'; ExternalVisible := 'False'; ExternalWritable := 'False'; } : BOOL;   //EPICS Status variable: GroupAlarm
      "Position_Discrep" { ExternalAccessible := 'True'; ExternalVisible := 'False'; ExternalWritable := 'False'; } : BOOL;   //EPICS Status variable: Position_Discrep
      "IO_Error" { ExternalAccessible := 'True'; ExternalVisible := 'False'; ExternalWritable := 'False'; } : BOOL;   //EPICS Status variable: IO_Error
      "Module_Error" { ExternalAccessible := 'True'; ExternalVisible := 'False'; ExternalWritable := 'False'; } : BOOL;   //EPICS Status variable: Module_Error
      "Input_Module_Error" { ExternalAccessible := 'True'; ExternalVisible := 'False'; ExternalWritable := 'False'; } : BOOL;   //EPICS Status variable: Input_Module_Error
      "Output_Module_Error" { ExternalAccessible := 'True'; ExternalVisible := 'False'; ExternalWritable := 'False'; } : BOOL;   //EPICS Status variable: Output_Module_Error
      "SPLimitActive" { ExternalAccessible := 'True'; ExternalVisible := 'False'; ExternalWritable := 'False'; } : BOOL;   //EPICS Status variable: SPLimitActive
      "SSTriggered" { ExternalAccessible := 'True'; ExternalVisible := 'False'; ExternalWritable := 'False'; } : BOOL;   //EPICS Status variable: SSTriggered
      "DiscrPerc" { ExternalAccessible := 'True'; ExternalVisible := 'False'; ExternalWritable := 'False'; } : REAL;   //EPICS Status variable: DiscrPerc
      "DiscrTime" { ExternalAccessible := 'True'; ExternalVisible := 'False'; ExternalWritable := 'False'; } : TIME;   //EPICS Status variable: DiscrTime
      "MaxRampUPSpd" { ExternalAccessible := 'True'; ExternalVisible := 'False'; ExternalWritable := 'False'; } : REAL;   //EPICS Status variable: MaxRampUPSpd
      "MaxRampDNSpd" { ExternalAccessible := 'True'; ExternalVisible := 'False'; ExternalWritable := 'False'; } : REAL;   //EPICS Status variable: MaxRampDNSpd
      "ActRampSpeed" { ExternalAccessible := 'True'; ExternalVisible := 'False'; ExternalWritable := 'False'; } : REAL;   //EPICS Status variable: ActRampSpeed
      "Ramping" { ExternalAccessible := 'True'; ExternalVisible := 'False'; ExternalWritable := 'False'; } : BOOL;   //EPICS Status variable: Ramping
      "RampSettingOK" { ExternalAccessible := 'True'; ExternalVisible := 'False'; ExternalWritable := 'False'; } : BOOL;   //EPICS Status variable: RampSettingOK
      "FB_RampUPTIME" { ExternalAccessible := 'True'; ExternalVisible := 'False'; ExternalWritable := 'False'; } : INT;   //EPICS Status variable: FB_RampUPTIME
      "FB_RampUPRANGE" { ExternalAccessible := 'True'; ExternalVisible := 'False'; ExternalWritable := 'False'; } : REAL;   //EPICS Status variable: FB_RampUPRANGE
      "FB_RampDNTIME" { ExternalAccessible := 'True'; ExternalVisible := 'False'; ExternalWritable := 'False'; } : INT;   //EPICS Status variable: FB_RampDNTIME
      "FB_RampDNRANGE" { ExternalAccessible := 'True'; ExternalVisible := 'False'; ExternalWritable := 'False'; } : REAL;   //EPICS Status variable: FB_RampDNRANGE
      "FB_ForcePosition" { ExternalAccessible := 'True'; ExternalVisible := 'False'; ExternalWritable := 'False'; } : REAL;   //EPICS Status variable: FB_ForcePosition
      "FB_Setpoint" { ExternalAccessible := 'True'; ExternalVisible := 'False'; ExternalWritable := 'False'; } : REAL;   //EPICS Status variable: FB_Setpoint
      "FB_Manipulated" { ExternalAccessible := 'True'; ExternalVisible := 'False'; ExternalWritable := 'False'; } : REAL;   //EPICS Status variable: FB_Manipulated
      "FB_Step" { ExternalAccessible := 'True'; ExternalVisible := 'False'; ExternalWritable := 'False'; } : REAL;   //EPICS Status variable: FB_Step
      "FB_RampTIME" { ExternalAccessible := 'True'; ExternalVisible := 'False'; ExternalWritable := 'False'; } : INT;   //EPICS Status variable: FB_RampTIME
      "FB_RampRANGE" { ExternalAccessible := 'True'; ExternalVisible := 'False'; ExternalWritable := 'False'; } : REAL;   //EPICS Status variable: FB_RampRANGE
      "Timer_enabled" { ExternalAccessible := 'True'; ExternalVisible := 'False'; ExternalWritable := 'False'; } : BOOL;   //EPICS Status variable: Timer_enabled
      "T_triggered" { ExternalAccessible := 'True'; ExternalVisible := 'False'; ExternalWritable := 'False'; } : BOOL;   //EPICS Status variable: T_triggered
      "T_running" { ExternalAccessible := 'True'; ExternalVisible := 'False'; ExternalWritable := 'False'; } : INT;   //EPICS Status variable: T_running
      "F_enabled" { ExternalAccessible := 'True'; ExternalVisible := 'False'; ExternalWritable := 'False'; } : BOOL;   //EPICS Status variable: F_enabled
      "FiltedValue" { ExternalAccessible := 'True'; ExternalVisible := 'False'; ExternalWritable := 'False'; } : REAL;   //EPICS Status variable: FiltedValue
   EPICSToPLCLength { ExternalAccessible := 'False'; ExternalVisible := 'False'; ExternalWritable := 'False'; } : Int;   // Length of device command register array (in words)
   EPICSToPLCDataBlockOffset { ExternalAccessible := 'False'; ExternalVisible := 'False'; ExternalWritable := 'False'; } : Int;   // Offset in EPICS->PLC comms block where this device data resides (in words)
   PLCToEPICSLength { ExternalAccessible := 'False'; ExternalVisible := 'False'; ExternalWritable := 'False'; } : Int;   // Length of device status register array (in words)
   PLCToEPICSDataBlockOffset { ExternalAccessible := 'False'; ExternalVisible := 'False'; ExternalWritable := 'False'; } : Int;   // Offset in PLC->EPICS comms block where this device data resides (in words)
   END_VAR
   VAR_OUTPUT
      "Cmd_Auto" { ExternalAccessible := 'True'; ExternalVisible := 'False'; ExternalWritable := 'False'; } : BOOL;   //EPICS Command variable: Cmd_Auto
      "Cmd_Manual" { ExternalAccessible := 'True'; ExternalVisible := 'False'; ExternalWritable := 'False'; } : BOOL;   //EPICS Command variable: Cmd_Manual
      "Cmd_Force" { ExternalAccessible := 'True'; ExternalVisible := 'False'; ExternalWritable := 'False'; } : BOOL;   //EPICS Command variable: Cmd_Force
      "Cmd_RampON" { ExternalAccessible := 'True'; ExternalVisible := 'False'; ExternalWritable := 'False'; } : BOOL;   //EPICS Command variable: Cmd_RampON
      "Cmd_RampOFF" { ExternalAccessible := 'True'; ExternalVisible := 'False'; ExternalWritable := 'False'; } : BOOL;   //EPICS Command variable: Cmd_RampOFF
      "Cmd_AckAlarm" { ExternalAccessible := 'True'; ExternalVisible := 'False'; ExternalWritable := 'False'; } : BOOL;   //EPICS Command variable: Cmd_AckAlarm
      "Cmd_ForceValInp" { ExternalAccessible := 'True'; ExternalVisible := 'False'; ExternalWritable := 'False'; } : BOOL;   //EPICS Command variable: Cmd_ForceValInp
      "Cmd_ForceValOut" { ExternalAccessible := 'True'; ExternalVisible := 'False'; ExternalWritable := 'False'; } : BOOL;   //EPICS Command variable: Cmd_ForceValOut
      "Cmd_ForceUnlock" { ExternalAccessible := 'True'; ExternalVisible := 'False'; ExternalWritable := 'False'; } : BOOL;   //EPICS Command variable: Cmd_ForceUnlock
      "Cmd_DevLock" { ExternalAccessible := 'True'; ExternalVisible := 'False'; ExternalWritable := 'False'; } : BOOL;   //EPICS Command variable: Cmd_DevLock
      "Cmd_DevUnlock" { ExternalAccessible := 'True'; ExternalVisible := 'False'; ExternalWritable := 'False'; } : BOOL;   //EPICS Command variable: Cmd_DevUnlock
      "P_ForcePosition" { ExternalAccessible := 'True'; ExternalVisible := 'False'; ExternalWritable := 'False'; } : REAL;   //EPICS Parameter variable: P_ForcePosition
      "P_Setpoint" { ExternalAccessible := 'True'; ExternalVisible := 'False'; ExternalWritable := 'False'; } : REAL;   //EPICS Parameter variable: P_Setpoint
      "P_Manipulated" { ExternalAccessible := 'True'; ExternalVisible := 'False'; ExternalWritable := 'False'; } : REAL;   //EPICS Parameter variable: P_Manipulated
      "P_Step" { ExternalAccessible := 'True'; ExternalVisible := 'False'; ExternalWritable := 'False'; } : REAL;   //EPICS Parameter variable: P_Step
      "P_RampUPTIME" { ExternalAccessible := 'True'; ExternalVisible := 'False'; ExternalWritable := 'False'; } : INT;   //EPICS Parameter variable: P_RampUPTIME
      "P_RampUPRANGE" { ExternalAccessible := 'True'; ExternalVisible := 'False'; ExternalWritable := 'False'; } : REAL;   //EPICS Parameter variable: P_RampUPRANGE
      "P_RampDNTIME" { ExternalAccessible := 'True'; ExternalVisible := 'False'; ExternalWritable := 'False'; } : INT;   //EPICS Parameter variable: P_RampDNTIME
      "P_RampDNRANGE" { ExternalAccessible := 'True'; ExternalVisible := 'False'; ExternalWritable := 'False'; } : REAL;   //EPICS Parameter variable: P_RampDNRANGE
      "P_Faceplate_LockID" { ExternalAccessible := 'True'; ExternalVisible := 'False'; ExternalWritable := 'False'; } : DINT;   //EPICS Parameter variable: P_Faceplate_LockID
      "P_BlockIcon_LockID" { ExternalAccessible := 'True'; ExternalVisible := 'False'; ExternalWritable := 'False'; } : DINT;   //EPICS Parameter variable: P_BlockIcon_LockID
      "T_period" { ExternalAccessible := 'True'; ExternalVisible := 'False'; ExternalWritable := 'False'; } : INT;   //EPICS Parameter variable: T_period
      "F_interval" { ExternalAccessible := 'True'; ExternalVisible := 'False'; ExternalWritable := 'False'; } : INT;   //EPICS Parameter variable: F_interval
      "F_buffer" { ExternalAccessible := 'True'; ExternalVisible := 'False'; ExternalWritable := 'False'; } : INT;   //EPICS Parameter variable: F_buffer
      "F_Enable" { ExternalAccessible := 'True'; ExternalVisible := 'False'; ExternalWritable := 'False'; } : BOOL;   //EPICS Parameter variable: F_Enable
      DEVICE_PARAM_OK { ExternalAccessible := 'False'; ExternalVisible := 'False'; ExternalWritable := 'False'; } : Bool;
   END_VAR
   VAR_IN_OUT
   END_VAR
   Var DB_SPECIFIC
      MyWord { ExternalAccessible := 'False'; ExternalVisible := 'False'; ExternalWritable := 'False'; } : Word;
      MyBytesinWord { ExternalAccessible := 'False'; ExternalVisible := 'False'; ExternalWritable := 'False'; } AT MyWord : Array[0..1] of Byte;
      MyBoolsinWord { ExternalAccessible := 'False'; ExternalVisible := 'False'; ExternalWritable := 'False'; } AT MyWord : Array[0..15] of Bool;
      MyDInt { ExternalAccessible := 'False'; ExternalVisible := 'False'; ExternalWritable := 'False'; } : DInt;
      MyWordsinDint { ExternalAccessible := 'False'; ExternalVisible := 'False'; ExternalWritable := 'False'; } AT MyDInt : Array[0..1] of Word;
      MyReal { ExternalAccessible := 'False'; ExternalVisible := 'False'; ExternalWritable := 'False'; } : Real;
      MyWordsinReal { ExternalAccessible := 'False'; ExternalVisible := 'False'; ExternalWritable := 'False'; } AT MyReal : Array[0..1] of Word;
      MyInt { ExternalAccessible := 'False'; ExternalVisible := 'False'; ExternalWritable := 'False'; } : Int;
      MyWordinInt { ExternalAccessible := 'False'; ExternalVisible := 'False'; ExternalWritable := 'False'; } AT MyInt : Word;
      MyDWord { ExternalAccessible := 'False'; ExternalVisible := 'False'; ExternalWritable := 'False'; } : DWord;
      MyWordsinDWord { ExternalAccessible := 'False'; ExternalVisible := 'False'; ExternalWritable := 'False'; } AT MyDWord : Array[0..1] of Word;
      MyTime { ExternalAccessible := 'False'; ExternalVisible := 'False'; ExternalWritable := 'False'; } : Time;
      MyWordsinTime { ExternalAccessible := 'False'; ExternalVisible := 'False'; ExternalWritable := 'False'; } AT MyTime : Array[0..1] of Word;
      MyString { ExternalAccessible := 'False'; ExternalVisible := 'False'; ExternalWritable := 'False'; } : String[40];
      MyWordsinString { ExternalAccessible := 'False'; ExternalVisible := 'False'; ExternalWritable := 'False'; } AT MyString : Array[0..20] of Word;
   END_VAR
   VAR_TEMP
      HashModbus : DInt;
      HashIFA : DInt;
      HashTIAMap : DInt;
      i : Int;
   END_VAR
    //Author: Miklos Boros (miklos.boros@esss.se), Copyrigth 2017-2020 by European Spallation Source, Lund
    //This block was generated by PLCFactory, please don't change it MANUALLY!
    //Input File Name: Spk-000CDL_Cryo-PLC-010-template-IFA-20220922093722.ifa
    //Generated: 20220922093722
    //According to HASH: 457744924
    //Device type: ICS_CV_PB_SIPART
    //Description: This function does the variable mapping for a device. All device-variable will be linked to an interface variable defined in this block.

    //********************************************
    //****************HASH check******************
    //********************************************


    #MyWordsinDint[0] := "EPICSToPLC"."Word"[0];
    #MyWordsinDint[1] := "EPICSToPLC"."Word"[1];
    #HashModbus := #MyDInt; //Hash from EPICS/ModbusTCP

    #HashIFA := 457744924; //Hash from Interface Factory as a constant

    #MyWordsinDint[0] := "PLCToEPICS"."Word"[0];
    #MyWordsinDint[1] := "PLCToEPICS"."Word"[1];
    #HashTIAMap := #MyDInt; //Hash from PLCFactory TIA Map


    IF ((#HashIFA = #HashModbus) AND (#HashModbus = #HashTIAMap)) THEN //Check CRCs
        #DEVICE_PARAM_OK := TRUE;
       //##################################### ICS HWI ###############################################
       //############################  ICS Instrument Library     ####################################
       //#  PLC Sample Code in VersionDog: ICS_LIBRARY_MASTER_PLC                                   ##
       //#  CCDB device types: ICS_CV_PB_SIPART                                                           ##
       //#  EPICS HMI (Block Icons/Faceplates)@ GitLab. Projekt: Cryo / CryogenicsLibrary / CryoLib ##
       //#                                                                                          ##
       //Siemens Sipart PS2 Valve Positioner
       //#                                                                                          ##
       //#
       //###########################           Version: 1.7           ################################
       //Author:	Emilio Asensi
       //Date:		06-09-2022
       //Version:  v1.7
       //Changes:
       //Added pvs for timer and filter
       //###########################           Version: 1.6           ################################
       //Author:	Emilio Asensi
       //Date:		03-05-2021
       //Version:  v1.6
       //Changes:
       //Added missing alarm signals                                                                                  ##
       //###########################           Version: 1.5           ################################
       //Author:	Peter Talas
       //Date:		16-03-2021
       //Version:  v1.5
       //Changes:
       //Archiving added
       //rpm changed to % on the ramping parameters
       //Interlock Message added
       //###########################           Version: 1.4           ################################
       //Author:	Miklos Boros
       //Date:		27-05-2019
       //Version:  v1.4
       //Changes:
       //Integration to CryoLibrary
       //Variable name unification
       //###########################           Version: 1.3           ################################
       //Author:	Emilio Asensi
       //Date:		24-01-2019
       //Version:  v1.3
       //Changes:
       //Accommodate changes on CMS_CV
       //1. Changed smoother ramping
       //Sipart module information
       //2. Removed Cascade operation
       //3. Modified CheckBack diagnostic bytes
       //###########################           Version: 1.2           ################################
       //Author:	Emilio Asensi
       //Date:		13-09-2018
       //Version:  v1.2
       //Changes:
       //Accommodate the changes on CMS_CV
       //1. Modified "For OPI visualisation" section: Added digital variable "FB_Keep_Setpoint".
       //2. Modified "Parameter Block" section: Added digital variable "P_Keep_Setpoint".
       //3. Modified Alarm Signal section to be compatible with new format.
       //###########################           Version: 1.0           ################################
       //Author:   Miklos Boros, Emilio Asensi
       //Date:	    17-05-2018
       //Version:  v1.0
       //Note:     Based on CMS_CV.def
       //#############################################################################################
       //###########################
       //STATUS BLOCK
       //###########################
       //Operation modes
       //OPI buttons
       //Setpoint and Manipulated value from HMI

    //********************************************
    //*************STATUS VARIABLES***************
    //********************************************


       #MyWord := W#0;
       #MyBoolsinWord[8] := #"OpMode_Auto";    //EPICSName: OpMode_Auto
       #MyBoolsinWord[9] := #"OpMode_Manual";    //EPICSName: OpMode_Manual
       #MyBoolsinWord[10] := #"OpMode_Forced";    //EPICSName: OpMode_Forced
       "PLCToEPICS"."Word"[#PLCToEPICSDataBlockOffset + 0] := #MyWord;

       #MyInt := #"ValveColor";    //EPICSName: ValveColor
       "PLCToEPICS"."Word"[#PLCToEPICSDataBlockOffset + 1] := #MyWordinInt;

       #MyReal := #"ValvePosition";    //EPICSName: ValvePosition
       "PLCToEPICS"."Word"[#PLCToEPICSDataBlockOffset + 2] := #MyWordsinReal[0];
       "PLCToEPICS"."Word"[#PLCToEPICSDataBlockOffset + 3] := #MyWordsinReal[1];

       #MyReal := #"ValveSP";    //EPICSName: ValveSP
       "PLCToEPICS"."Word"[#PLCToEPICSDataBlockOffset + 4] := #MyWordsinReal[0];
       "PLCToEPICS"."Word"[#PLCToEPICSDataBlockOffset + 5] := #MyWordsinReal[1];

       #MyReal := #"ValveMV";    //EPICSName: ValveMV
       "PLCToEPICS"."Word"[#PLCToEPICSDataBlockOffset + 6] := #MyWordsinReal[0];
       "PLCToEPICS"."Word"[#PLCToEPICSDataBlockOffset + 7] := #MyWordsinReal[1];

       #MyWord := W#0;
       #MyBoolsinWord[8] := #"Opening";    //EPICSName: Opening
       #MyBoolsinWord[9] := #"Closing";    //EPICSName: Closing
       "PLCToEPICS"."Word"[#PLCToEPICSDataBlockOffset + 8] := #MyWord;

       #MyWord := W#0;
       #MyBytesinWord[0] := #"StatusRB";    //EPICSName: StatusRB
       "PLCToEPICS"."Word"[#PLCToEPICSDataBlockOffset + 9] := #MyWord;

       #MyInt := #"DiscretePosition";    //EPICSName: DiscretePosition
       "PLCToEPICS"."Word"[#PLCToEPICSDataBlockOffset + 10] := #MyWordinInt;

       #MyWord := W#0;
       #MyBytesinWord[0] := #"DiscreteStatus";    //EPICSName: DiscreteStatus
       "PLCToEPICS"."Word"[#PLCToEPICSDataBlockOffset + 11] := #MyWord;

       #MyWord := W#0;
       #MyBytesinWord[0] := #"DiagnosticsCB01";    //EPICSName: DiagnosticsCB01
       "PLCToEPICS"."Word"[#PLCToEPICSDataBlockOffset + 12] := #MyWord;

       #MyWord := W#0;
       #MyBytesinWord[0] := #"DiagnosticsCB02";    //EPICSName: DiagnosticsCB02
       "PLCToEPICS"."Word"[#PLCToEPICSDataBlockOffset + 13] := #MyWord;

       #MyWord := W#0;
       #MyBytesinWord[0] := #"DiagnosticsCB03";    //EPICSName: DiagnosticsCB03
       "PLCToEPICS"."Word"[#PLCToEPICSDataBlockOffset + 14] := #MyWord;

       #MyWord := W#0;
       #MyBoolsinWord[8] := #"Inhibit_Manual";    //EPICSName: Inhibit_Manual
       #MyBoolsinWord[9] := #"Inhibit_Force";    //EPICSName: Inhibit_Force
       #MyBoolsinWord[10] := #"Inhibit_Lock";    //EPICSName: Inhibit_Lock
       #MyBoolsinWord[11] := #"GroupInterlock";    //EPICSName: GroupInterlock
       "PLCToEPICS"."Word"[#PLCToEPICSDataBlockOffset + 15] := #MyWord;

       // Clear the buffer of any residual data, but skip the first word as that is the actual and maximum length
       FOR #i:=1 TO 20 DO
            #MyWordsinString[#i] := 0;
       END_FOR;
       #MyString := #"InterlockMsg";  //EPICSName: InterlockMsg
       FOR #i:=0 TO 18 DO
            "PLCToEPICS"."Word"[#PLCToEPICSDataBlockOffset + 16 + #i] := #MyWordsinString[#i + 1];
       END_FOR;
       // Terminate C-string
       "PLCToEPICS"."Word"[#PLCToEPICSDataBlockOffset + 16 + 19] := #MyWordsinString[20] & 16#FF00;

       #MyWord := W#0;
       #MyBoolsinWord[8] := #"MoveInterlock";    //EPICSName: MoveInterlock
       #MyBoolsinWord[9] := #"EnableAutoBtn";    //EPICSName: EnableAutoBtn
       #MyBoolsinWord[10] := #"EnableManualBtn";    //EPICSName: EnableManualBtn
       #MyBoolsinWord[11] := #"EnableForcedBtn";    //EPICSName: EnableForcedBtn
       #MyBoolsinWord[12] := #"EnableBlkCtrl";    //EPICSName: EnableBlkCtrl
       #MyBoolsinWord[13] := #"EnableForceValBtn";    //EPICSName: EnableForceValBtn
       #MyBoolsinWord[14] := #"DevLocked";    //EPICSName: DevLocked
       "PLCToEPICS"."Word"[#PLCToEPICSDataBlockOffset + 36] := #MyWord;

       #MyDInt := #"Faceplate_LockID";    //EPICSName: Faceplate_LockID
       "PLCToEPICS"."Word"[#PLCToEPICSDataBlockOffset + 37] := #MyWordsinDint[0];
       "PLCToEPICS"."Word"[#PLCToEPICSDataBlockOffset + 38] := #MyWordsinDint[1];

       #MyDInt := #"BlockIcon_LockID";    //EPICSName: BlockIcon_LockID
       "PLCToEPICS"."Word"[#PLCToEPICSDataBlockOffset + 39] := #MyWordsinDint[0];
       "PLCToEPICS"."Word"[#PLCToEPICSDataBlockOffset + 40] := #MyWordsinDint[1];

       #MyWord := W#0;
       #MyBoolsinWord[8] := #"LatchAlarm";    //EPICSName: LatchAlarm
       #MyBoolsinWord[9] := #"GroupAlarm";    //EPICSName: GroupAlarm
       #MyBoolsinWord[10] := #"Position_Discrep";    //EPICSName: Position_Discrep
       #MyBoolsinWord[11] := #"IO_Error";    //EPICSName: IO_Error
       #MyBoolsinWord[12] := #"Module_Error";    //EPICSName: Module_Error
       #MyBoolsinWord[13] := #"Input_Module_Error";    //EPICSName: Input_Module_Error
       #MyBoolsinWord[14] := #"Output_Module_Error";    //EPICSName: Output_Module_Error
       #MyBoolsinWord[15] := #"SPLimitActive";    //EPICSName: SPLimitActive
       #MyBoolsinWord[0] := #"SSTriggered";    //EPICSName: SSTriggered
       "PLCToEPICS"."Word"[#PLCToEPICSDataBlockOffset + 41] := #MyWord;

       #MyReal := #"DiscrPerc";    //EPICSName: DiscrPerc
       "PLCToEPICS"."Word"[#PLCToEPICSDataBlockOffset + 42] := #MyWordsinReal[0];
       "PLCToEPICS"."Word"[#PLCToEPICSDataBlockOffset + 43] := #MyWordsinReal[1];

       #MyTime := #"DiscrTime";    //EPICSName: DiscrTime
       "PLCToEPICS"."Word"[#PLCToEPICSDataBlockOffset + 44] := #MyWordsinTime[0];
       "PLCToEPICS"."Word"[#PLCToEPICSDataBlockOffset + 45] := #MyWordsinTime[1];

       #MyReal := #"MaxRampUPSpd";    //EPICSName: MaxRampUPSpd
       "PLCToEPICS"."Word"[#PLCToEPICSDataBlockOffset + 46] := #MyWordsinReal[0];
       "PLCToEPICS"."Word"[#PLCToEPICSDataBlockOffset + 47] := #MyWordsinReal[1];

       #MyReal := #"MaxRampDNSpd";    //EPICSName: MaxRampDNSpd
       "PLCToEPICS"."Word"[#PLCToEPICSDataBlockOffset + 48] := #MyWordsinReal[0];
       "PLCToEPICS"."Word"[#PLCToEPICSDataBlockOffset + 49] := #MyWordsinReal[1];

       #MyReal := #"ActRampSpeed";    //EPICSName: ActRampSpeed
       "PLCToEPICS"."Word"[#PLCToEPICSDataBlockOffset + 50] := #MyWordsinReal[0];
       "PLCToEPICS"."Word"[#PLCToEPICSDataBlockOffset + 51] := #MyWordsinReal[1];

       #MyWord := W#0;
       #MyBoolsinWord[8] := #"Ramping";    //EPICSName: Ramping
       #MyBoolsinWord[9] := #"RampSettingOK";    //EPICSName: RampSettingOK
       "PLCToEPICS"."Word"[#PLCToEPICSDataBlockOffset + 52] := #MyWord;

       #MyInt := #"FB_RampUPTIME";    //EPICSName: FB_RampUPTIME
       "PLCToEPICS"."Word"[#PLCToEPICSDataBlockOffset + 53] := #MyWordinInt;

       #MyReal := #"FB_RampUPRANGE";    //EPICSName: FB_RampUPRANGE
       "PLCToEPICS"."Word"[#PLCToEPICSDataBlockOffset + 54] := #MyWordsinReal[0];
       "PLCToEPICS"."Word"[#PLCToEPICSDataBlockOffset + 55] := #MyWordsinReal[1];

       #MyInt := #"FB_RampDNTIME";    //EPICSName: FB_RampDNTIME
       "PLCToEPICS"."Word"[#PLCToEPICSDataBlockOffset + 56] := #MyWordinInt;

       #MyReal := #"FB_RampDNRANGE";    //EPICSName: FB_RampDNRANGE
       "PLCToEPICS"."Word"[#PLCToEPICSDataBlockOffset + 57] := #MyWordsinReal[0];
       "PLCToEPICS"."Word"[#PLCToEPICSDataBlockOffset + 58] := #MyWordsinReal[1];

       #MyReal := #"FB_ForcePosition";    //EPICSName: FB_ForcePosition
       "PLCToEPICS"."Word"[#PLCToEPICSDataBlockOffset + 59] := #MyWordsinReal[0];
       "PLCToEPICS"."Word"[#PLCToEPICSDataBlockOffset + 60] := #MyWordsinReal[1];

       #MyReal := #"FB_Setpoint";    //EPICSName: FB_Setpoint
       "PLCToEPICS"."Word"[#PLCToEPICSDataBlockOffset + 61] := #MyWordsinReal[0];
       "PLCToEPICS"."Word"[#PLCToEPICSDataBlockOffset + 62] := #MyWordsinReal[1];

       #MyReal := #"FB_Manipulated";    //EPICSName: FB_Manipulated
       "PLCToEPICS"."Word"[#PLCToEPICSDataBlockOffset + 63] := #MyWordsinReal[0];
       "PLCToEPICS"."Word"[#PLCToEPICSDataBlockOffset + 64] := #MyWordsinReal[1];

       #MyReal := #"FB_Step";    //EPICSName: FB_Step
       "PLCToEPICS"."Word"[#PLCToEPICSDataBlockOffset + 65] := #MyWordsinReal[0];
       "PLCToEPICS"."Word"[#PLCToEPICSDataBlockOffset + 66] := #MyWordsinReal[1];

       #MyInt := #"FB_RampTIME";    //EPICSName: FB_RampTIME
       "PLCToEPICS"."Word"[#PLCToEPICSDataBlockOffset + 67] := #MyWordinInt;

       #MyReal := #"FB_RampRANGE";    //EPICSName: FB_RampRANGE
       "PLCToEPICS"."Word"[#PLCToEPICSDataBlockOffset + 68] := #MyWordsinReal[0];
       "PLCToEPICS"."Word"[#PLCToEPICSDataBlockOffset + 69] := #MyWordsinReal[1];

       #MyWord := W#0;
       #MyBoolsinWord[8] := #"Timer_enabled";    //EPICSName: Timer_enabled
       #MyBoolsinWord[9] := #"T_triggered";    //EPICSName: T_triggered
       "PLCToEPICS"."Word"[#PLCToEPICSDataBlockOffset + 70] := #MyWord;

       #MyInt := #"T_running";    //EPICSName: T_running
       "PLCToEPICS"."Word"[#PLCToEPICSDataBlockOffset + 71] := #MyWordinInt;

       #MyWord := W#0;
       #MyBoolsinWord[8] := #"F_enabled";    //EPICSName: F_enabled
       "PLCToEPICS"."Word"[#PLCToEPICSDataBlockOffset + 72] := #MyWord;

       #MyReal := #"FiltedValue";    //EPICSName: FiltedValue
       "PLCToEPICS"."Word"[#PLCToEPICSDataBlockOffset + 73] := #MyWordsinReal[0];
       "PLCToEPICS"."Word"[#PLCToEPICSDataBlockOffset + 74] := #MyWordsinReal[1];

    //********************************************
    //*************COMMAND VARIABLES**************
    //********************************************


       #MyWord := "EPICSToPLC"."Word"[#EPICSToPLCDataBlockOffset + 0];
       "EPICSToPLC"."Word"[#EPICSToPLCDataBlockOffset + 0] := 0;
       #"Cmd_Auto" := #MyBoolsinWord[8];    //EPICSName: Cmd_Auto
       #"Cmd_Manual" := #MyBoolsinWord[9];    //EPICSName: Cmd_Manual
       #"Cmd_Force" := #MyBoolsinWord[10];    //EPICSName: Cmd_Force
       #"Cmd_RampON" := #MyBoolsinWord[11];    //EPICSName: Cmd_RampON
       #"Cmd_RampOFF" := #MyBoolsinWord[12];    //EPICSName: Cmd_RampOFF
       #"Cmd_AckAlarm" := #MyBoolsinWord[13];    //EPICSName: Cmd_AckAlarm
       #"Cmd_ForceValInp" := #MyBoolsinWord[14];    //EPICSName: Cmd_ForceValInp
       #"Cmd_ForceValOut" := #MyBoolsinWord[15];    //EPICSName: Cmd_ForceValOut
       #"Cmd_ForceUnlock" := #MyBoolsinWord[0];    //EPICSName: Cmd_ForceUnlock
       #"Cmd_DevLock" := #MyBoolsinWord[1];    //EPICSName: Cmd_DevLock
       #"Cmd_DevUnlock" := #MyBoolsinWord[2];    //EPICSName: Cmd_DevUnlock

    //********************************************
    //************PARAMETER VARIABLES*************
    //********************************************


       #MyReal	:= 0.0;
       #MyWordsinReal[0]	:= "EPICSToPLC"."Word"[#EPICSToPLCDataBlockOffset + 1];
       #MyWordsinReal[1]	:= "EPICSToPLC"."Word"[#EPICSToPLCDataBlockOffset + 2];
       #"P_ForcePosition" := #MyReal;    //EPICSName: P_ForcePosition

       #MyReal	:= 0.0;
       #MyWordsinReal[0]	:= "EPICSToPLC"."Word"[#EPICSToPLCDataBlockOffset + 3];
       #MyWordsinReal[1]	:= "EPICSToPLC"."Word"[#EPICSToPLCDataBlockOffset + 4];
       #"P_Setpoint" := #MyReal;    //EPICSName: P_Setpoint

       #MyReal	:= 0.0;
       #MyWordsinReal[0]	:= "EPICSToPLC"."Word"[#EPICSToPLCDataBlockOffset + 5];
       #MyWordsinReal[1]	:= "EPICSToPLC"."Word"[#EPICSToPLCDataBlockOffset + 6];
       #"P_Manipulated" := #MyReal;    //EPICSName: P_Manipulated

       #MyReal	:= 0.0;
       #MyWordsinReal[0]	:= "EPICSToPLC"."Word"[#EPICSToPLCDataBlockOffset + 7];
       #MyWordsinReal[1]	:= "EPICSToPLC"."Word"[#EPICSToPLCDataBlockOffset + 8];
       #"P_Step" := #MyReal;    //EPICSName: P_Step

       #MyWordinInt := "EPICSToPLC"."Word"[#EPICSToPLCDataBlockOffset + 9];
       #"P_RampUPTIME" := #MyInt;    //EPICSName: P_RampUPTIME

       #MyReal	:= 0.0;
       #MyWordsinReal[0]	:= "EPICSToPLC"."Word"[#EPICSToPLCDataBlockOffset + 10];
       #MyWordsinReal[1]	:= "EPICSToPLC"."Word"[#EPICSToPLCDataBlockOffset + 11];
       #"P_RampUPRANGE" := #MyReal;    //EPICSName: P_RampUPRANGE

       #MyWordinInt := "EPICSToPLC"."Word"[#EPICSToPLCDataBlockOffset + 12];
       #"P_RampDNTIME" := #MyInt;    //EPICSName: P_RampDNTIME

       #MyReal	:= 0.0;
       #MyWordsinReal[0]	:= "EPICSToPLC"."Word"[#EPICSToPLCDataBlockOffset + 13];
       #MyWordsinReal[1]	:= "EPICSToPLC"."Word"[#EPICSToPLCDataBlockOffset + 14];
       #"P_RampDNRANGE" := #MyReal;    //EPICSName: P_RampDNRANGE

       #MyDInt	:= 0;
       #MyWordsinDint[0]	:= "EPICSToPLC"."Word"[#EPICSToPLCDataBlockOffset + 15];
       #MyWordsinDint[1]	:= "EPICSToPLC"."Word"[#EPICSToPLCDataBlockOffset + 16];
       #"P_Faceplate_LockID" := #MyDInt;    //EPICSName: P_Faceplate_LockID

       #MyDInt	:= 0;
       #MyWordsinDint[0]	:= "EPICSToPLC"."Word"[#EPICSToPLCDataBlockOffset + 17];
       #MyWordsinDint[1]	:= "EPICSToPLC"."Word"[#EPICSToPLCDataBlockOffset + 18];
       #"P_BlockIcon_LockID" := #MyDInt;    //EPICSName: P_BlockIcon_LockID

       #MyWordinInt := "EPICSToPLC"."Word"[#EPICSToPLCDataBlockOffset + 19];
       #"T_period" := #MyInt;    //EPICSName: T_period

       #MyWordinInt := "EPICSToPLC"."Word"[#EPICSToPLCDataBlockOffset + 20];
       #"F_interval" := #MyInt;    //EPICSName: F_interval

       #MyWordinInt := "EPICSToPLC"."Word"[#EPICSToPLCDataBlockOffset + 21];
       #"F_buffer" := #MyInt;    //EPICSName: F_buffer

       #MyWord := "EPICSToPLC"."Word"[#EPICSToPLCDataBlockOffset + 22];
       #"F_Enable" := #MyBoolsinWord[8];    //EPICSName: F_Enable
    Else
       #DEVICE_PARAM_OK := FALSE; //Invalid Hash
    END_IF;
END_FUNCTION_BLOCK
FUNCTION_BLOCK "DEVTYPE_ICS_EH"
{ S7_Optimized_Access := 'TRUE' }
VERSION : 1.0
   VAR_INPUT
      "OpMode_Auto" { ExternalAccessible := 'True'; ExternalVisible := 'False'; ExternalWritable := 'False'; } : BOOL;   //EPICS Status variable: OpMode_Auto
      "OpMode_Manual" { ExternalAccessible := 'True'; ExternalVisible := 'False'; ExternalWritable := 'False'; } : BOOL;   //EPICS Status variable: OpMode_Manual
      "OpMode_Forced" { ExternalAccessible := 'True'; ExternalVisible := 'False'; ExternalWritable := 'False'; } : BOOL;   //EPICS Status variable: OpMode_Forced
      "HeaterCurrent" { ExternalAccessible := 'True'; ExternalVisible := 'False'; ExternalWritable := 'False'; } : REAL;   //EPICS Status variable: HeaterCurrent
      "HeaterVoltage" { ExternalAccessible := 'True'; ExternalVisible := 'False'; ExternalWritable := 'False'; } : REAL;   //EPICS Status variable: HeaterVoltage
      "HeaterPower" { ExternalAccessible := 'True'; ExternalVisible := 'False'; ExternalWritable := 'False'; } : REAL;   //EPICS Status variable: HeaterPower
      "HeaterSP" { ExternalAccessible := 'True'; ExternalVisible := 'False'; ExternalWritable := 'False'; } : REAL;   //EPICS Status variable: HeaterSP
      "HeaterMV" { ExternalAccessible := 'True'; ExternalVisible := 'False'; ExternalWritable := 'False'; } : REAL;   //EPICS Status variable: HeaterMV
      "HeatingON" { ExternalAccessible := 'True'; ExternalVisible := 'False'; ExternalWritable := 'False'; } : BOOL;   //EPICS Status variable: HeatingON
      "Inhibit_Manual" { ExternalAccessible := 'True'; ExternalVisible := 'False'; ExternalWritable := 'False'; } : BOOL;   //EPICS Status variable: Inhibit_Manual
      "Inhibit_Force" { ExternalAccessible := 'True'; ExternalVisible := 'False'; ExternalWritable := 'False'; } : BOOL;   //EPICS Status variable: Inhibit_Force
      "Inhibit_Lock" { ExternalAccessible := 'True'; ExternalVisible := 'False'; ExternalWritable := 'False'; } : BOOL;   //EPICS Status variable: Inhibit_Lock
      "GroupInterlock" { ExternalAccessible := 'True'; ExternalVisible := 'False'; ExternalWritable := 'False'; } : BOOL;   //EPICS Status variable: GroupInterlock
      "HeatInterlock" { ExternalAccessible := 'True'; ExternalVisible := 'False'; ExternalWritable := 'False'; } : BOOL;   //EPICS Status variable: HeatInterlock
      "EnableAutoBtn" { ExternalAccessible := 'True'; ExternalVisible := 'False'; ExternalWritable := 'False'; } : BOOL;   //EPICS Status variable: EnableAutoBtn
      "EnableManualBtn" { ExternalAccessible := 'True'; ExternalVisible := 'False'; ExternalWritable := 'False'; } : BOOL;   //EPICS Status variable: EnableManualBtn
      "EnableForcedBtn" { ExternalAccessible := 'True'; ExternalVisible := 'False'; ExternalWritable := 'False'; } : BOOL;   //EPICS Status variable: EnableForcedBtn
      "EnableForceValBtn" { ExternalAccessible := 'True'; ExternalVisible := 'False'; ExternalWritable := 'False'; } : BOOL;   //EPICS Status variable: EnableForceValBtn
      "DevLocked" { ExternalAccessible := 'True'; ExternalVisible := 'False'; ExternalWritable := 'False'; } : BOOL;   //EPICS Status variable: DevLocked
      "Faceplate_LockID" { ExternalAccessible := 'True'; ExternalVisible := 'False'; ExternalWritable := 'False'; } : DINT;   //EPICS Status variable: Faceplate_LockID
      "BlockIcon_LockID" { ExternalAccessible := 'True'; ExternalVisible := 'False'; ExternalWritable := 'False'; } : DINT;   //EPICS Status variable: BlockIcon_LockID
      "LatchAlarm" { ExternalAccessible := 'True'; ExternalVisible := 'False'; ExternalWritable := 'False'; } : BOOL;   //EPICS Status variable: LatchAlarm
      "GroupAlarm" { ExternalAccessible := 'True'; ExternalVisible := 'False'; ExternalWritable := 'False'; } : BOOL;   //EPICS Status variable: GroupAlarm
      "Power_Discrep" { ExternalAccessible := 'True'; ExternalVisible := 'False'; ExternalWritable := 'False'; } : BOOL;   //EPICS Status variable: Power_Discrep
      "IO_Error" { ExternalAccessible := 'True'; ExternalVisible := 'False'; ExternalWritable := 'False'; } : BOOL;   //EPICS Status variable: IO_Error
      "Input_Module_Error" { ExternalAccessible := 'True'; ExternalVisible := 'False'; ExternalWritable := 'False'; } : BOOL;   //EPICS Status variable: Input_Module_Error
      "Output_Module_Error" { ExternalAccessible := 'True'; ExternalVisible := 'False'; ExternalWritable := 'False'; } : BOOL;   //EPICS Status variable: Output_Module_Error
      "DiscrPerc" { ExternalAccessible := 'True'; ExternalVisible := 'False'; ExternalWritable := 'False'; } : REAL;   //EPICS Status variable: DiscrPerc
      "DiscrTime" { ExternalAccessible := 'True'; ExternalVisible := 'False'; ExternalWritable := 'False'; } : TIME;   //EPICS Status variable: DiscrTime
      "MaxRampUPSpd" { ExternalAccessible := 'True'; ExternalVisible := 'False'; ExternalWritable := 'False'; } : REAL;   //EPICS Status variable: MaxRampUPSpd
      "MaxRampDNSpd" { ExternalAccessible := 'True'; ExternalVisible := 'False'; ExternalWritable := 'False'; } : REAL;   //EPICS Status variable: MaxRampDNSpd
      "ActRampSpeed" { ExternalAccessible := 'True'; ExternalVisible := 'False'; ExternalWritable := 'False'; } : REAL;   //EPICS Status variable: ActRampSpeed
      "Ramping" { ExternalAccessible := 'True'; ExternalVisible := 'False'; ExternalWritable := 'False'; } : BOOL;   //EPICS Status variable: Ramping
      "RampSettingOK" { ExternalAccessible := 'True'; ExternalVisible := 'False'; ExternalWritable := 'False'; } : BOOL;   //EPICS Status variable: RampSettingOK
      "FB_RampUPTIME" { ExternalAccessible := 'True'; ExternalVisible := 'False'; ExternalWritable := 'False'; } : INT;   //EPICS Status variable: FB_RampUPTIME
      "FB_RampUPRANGE" { ExternalAccessible := 'True'; ExternalVisible := 'False'; ExternalWritable := 'False'; } : REAL;   //EPICS Status variable: FB_RampUPRANGE
      "FB_RampDNTIME" { ExternalAccessible := 'True'; ExternalVisible := 'False'; ExternalWritable := 'False'; } : INT;   //EPICS Status variable: FB_RampDNTIME
      "FB_RampDNRANGE" { ExternalAccessible := 'True'; ExternalVisible := 'False'; ExternalWritable := 'False'; } : REAL;   //EPICS Status variable: FB_RampDNRANGE
      "FB_ForcePower" { ExternalAccessible := 'True'; ExternalVisible := 'False'; ExternalWritable := 'False'; } : REAL;   //EPICS Status variable: FB_ForcePower
      "FB_Setpoint" { ExternalAccessible := 'True'; ExternalVisible := 'False'; ExternalWritable := 'False'; } : REAL;   //EPICS Status variable: FB_Setpoint
      "FB_Manipulated" { ExternalAccessible := 'True'; ExternalVisible := 'False'; ExternalWritable := 'False'; } : REAL;   //EPICS Status variable: FB_Manipulated
      "FB_Step" { ExternalAccessible := 'True'; ExternalVisible := 'False'; ExternalWritable := 'False'; } : REAL;   //EPICS Status variable: FB_Step
      "FB_RampTIME" { ExternalAccessible := 'True'; ExternalVisible := 'False'; ExternalWritable := 'False'; } : INT;   //EPICS Status variable: FB_RampTIME
      "FB_RampRANGE" { ExternalAccessible := 'True'; ExternalVisible := 'False'; ExternalWritable := 'False'; } : REAL;   //EPICS Status variable: FB_RampRANGE
   EPICSToPLCLength { ExternalAccessible := 'False'; ExternalVisible := 'False'; ExternalWritable := 'False'; } : Int;   // Length of device command register array (in words)
   EPICSToPLCDataBlockOffset { ExternalAccessible := 'False'; ExternalVisible := 'False'; ExternalWritable := 'False'; } : Int;   // Offset in EPICS->PLC comms block where this device data resides (in words)
   PLCToEPICSLength { ExternalAccessible := 'False'; ExternalVisible := 'False'; ExternalWritable := 'False'; } : Int;   // Length of device status register array (in words)
   PLCToEPICSDataBlockOffset { ExternalAccessible := 'False'; ExternalVisible := 'False'; ExternalWritable := 'False'; } : Int;   // Offset in PLC->EPICS comms block where this device data resides (in words)
   END_VAR
   VAR_OUTPUT
      "Cmd_Auto" { ExternalAccessible := 'True'; ExternalVisible := 'False'; ExternalWritable := 'False'; } : BOOL;   //EPICS Command variable: Cmd_Auto
      "Cmd_Manual" { ExternalAccessible := 'True'; ExternalVisible := 'False'; ExternalWritable := 'False'; } : BOOL;   //EPICS Command variable: Cmd_Manual
      "Cmd_Force" { ExternalAccessible := 'True'; ExternalVisible := 'False'; ExternalWritable := 'False'; } : BOOL;   //EPICS Command variable: Cmd_Force
      "Cmd_RampON" { ExternalAccessible := 'True'; ExternalVisible := 'False'; ExternalWritable := 'False'; } : BOOL;   //EPICS Command variable: Cmd_RampON
      "Cmd_RampOFF" { ExternalAccessible := 'True'; ExternalVisible := 'False'; ExternalWritable := 'False'; } : BOOL;   //EPICS Command variable: Cmd_RampOFF
      "Cmd_AckAlarm" { ExternalAccessible := 'True'; ExternalVisible := 'False'; ExternalWritable := 'False'; } : BOOL;   //EPICS Command variable: Cmd_AckAlarm
      "Cmd_ForceValInp" { ExternalAccessible := 'True'; ExternalVisible := 'False'; ExternalWritable := 'False'; } : BOOL;   //EPICS Command variable: Cmd_ForceValInp
      "Cmd_ForceValOut" { ExternalAccessible := 'True'; ExternalVisible := 'False'; ExternalWritable := 'False'; } : BOOL;   //EPICS Command variable: Cmd_ForceValOut
      "Cmd_ForceUnlock" { ExternalAccessible := 'True'; ExternalVisible := 'False'; ExternalWritable := 'False'; } : BOOL;   //EPICS Command variable: Cmd_ForceUnlock
      "Cmd_DevLock" { ExternalAccessible := 'True'; ExternalVisible := 'False'; ExternalWritable := 'False'; } : BOOL;   //EPICS Command variable: Cmd_DevLock
      "Cmd_DevUnlock" { ExternalAccessible := 'True'; ExternalVisible := 'False'; ExternalWritable := 'False'; } : BOOL;   //EPICS Command variable: Cmd_DevUnlock
      "P_ForcePower" { ExternalAccessible := 'True'; ExternalVisible := 'False'; ExternalWritable := 'False'; } : REAL;   //EPICS Parameter variable: P_ForcePower
      "P_Setpoint" { ExternalAccessible := 'True'; ExternalVisible := 'False'; ExternalWritable := 'False'; } : REAL;   //EPICS Parameter variable: P_Setpoint
      "P_Manipulated" { ExternalAccessible := 'True'; ExternalVisible := 'False'; ExternalWritable := 'False'; } : REAL;   //EPICS Parameter variable: P_Manipulated
      "P_Step" { ExternalAccessible := 'True'; ExternalVisible := 'False'; ExternalWritable := 'False'; } : REAL;   //EPICS Parameter variable: P_Step
      "P_RampUPTIME" { ExternalAccessible := 'True'; ExternalVisible := 'False'; ExternalWritable := 'False'; } : INT;   //EPICS Parameter variable: P_RampUPTIME
      "P_RampUPRANGE" { ExternalAccessible := 'True'; ExternalVisible := 'False'; ExternalWritable := 'False'; } : REAL;   //EPICS Parameter variable: P_RampUPRANGE
      "P_RampDNTIME" { ExternalAccessible := 'True'; ExternalVisible := 'False'; ExternalWritable := 'False'; } : INT;   //EPICS Parameter variable: P_RampDNTIME
      "P_RampDNRANGE" { ExternalAccessible := 'True'; ExternalVisible := 'False'; ExternalWritable := 'False'; } : REAL;   //EPICS Parameter variable: P_RampDNRANGE
      "P_Faceplate_LockID" { ExternalAccessible := 'True'; ExternalVisible := 'False'; ExternalWritable := 'False'; } : DINT;   //EPICS Parameter variable: P_Faceplate_LockID
      "P_BlockIcon_LockID" { ExternalAccessible := 'True'; ExternalVisible := 'False'; ExternalWritable := 'False'; } : DINT;   //EPICS Parameter variable: P_BlockIcon_LockID
      DEVICE_PARAM_OK { ExternalAccessible := 'False'; ExternalVisible := 'False'; ExternalWritable := 'False'; } : Bool;
   END_VAR
   VAR_IN_OUT
   END_VAR
   Var DB_SPECIFIC
      MyWord { ExternalAccessible := 'False'; ExternalVisible := 'False'; ExternalWritable := 'False'; } : Word;
      MyBytesinWord { ExternalAccessible := 'False'; ExternalVisible := 'False'; ExternalWritable := 'False'; } AT MyWord : Array[0..1] of Byte;
      MyBoolsinWord { ExternalAccessible := 'False'; ExternalVisible := 'False'; ExternalWritable := 'False'; } AT MyWord : Array[0..15] of Bool;
      MyDInt { ExternalAccessible := 'False'; ExternalVisible := 'False'; ExternalWritable := 'False'; } : DInt;
      MyWordsinDint { ExternalAccessible := 'False'; ExternalVisible := 'False'; ExternalWritable := 'False'; } AT MyDInt : Array[0..1] of Word;
      MyReal { ExternalAccessible := 'False'; ExternalVisible := 'False'; ExternalWritable := 'False'; } : Real;
      MyWordsinReal { ExternalAccessible := 'False'; ExternalVisible := 'False'; ExternalWritable := 'False'; } AT MyReal : Array[0..1] of Word;
      MyInt { ExternalAccessible := 'False'; ExternalVisible := 'False'; ExternalWritable := 'False'; } : Int;
      MyWordinInt { ExternalAccessible := 'False'; ExternalVisible := 'False'; ExternalWritable := 'False'; } AT MyInt : Word;
      MyDWord { ExternalAccessible := 'False'; ExternalVisible := 'False'; ExternalWritable := 'False'; } : DWord;
      MyWordsinDWord { ExternalAccessible := 'False'; ExternalVisible := 'False'; ExternalWritable := 'False'; } AT MyDWord : Array[0..1] of Word;
      MyTime { ExternalAccessible := 'False'; ExternalVisible := 'False'; ExternalWritable := 'False'; } : Time;
      MyWordsinTime { ExternalAccessible := 'False'; ExternalVisible := 'False'; ExternalWritable := 'False'; } AT MyTime : Array[0..1] of Word;
      MyString { ExternalAccessible := 'False'; ExternalVisible := 'False'; ExternalWritable := 'False'; } : String[40];
      MyWordsinString { ExternalAccessible := 'False'; ExternalVisible := 'False'; ExternalWritable := 'False'; } AT MyString : Array[0..20] of Word;
   END_VAR
   VAR_TEMP
      HashModbus : DInt;
      HashIFA : DInt;
      HashTIAMap : DInt;
      i : Int;
   END_VAR
    //Author: Miklos Boros (miklos.boros@esss.se), Copyrigth 2017-2020 by European Spallation Source, Lund
    //This block was generated by PLCFactory, please don't change it MANUALLY!
    //Input File Name: Spk-000CDL_Cryo-PLC-010-template-IFA-20220922093722.ifa
    //Generated: 20220922093722
    //According to HASH: 457744924
    //Device type: ICS_EH
    //Description: This function does the variable mapping for a device. All device-variable will be linked to an interface variable defined in this block.

    //********************************************
    //****************HASH check******************
    //********************************************


    #MyWordsinDint[0] := "EPICSToPLC"."Word"[0];
    #MyWordsinDint[1] := "EPICSToPLC"."Word"[1];
    #HashModbus := #MyDInt; //Hash from EPICS/ModbusTCP

    #HashIFA := 457744924; //Hash from Interface Factory as a constant

    #MyWordsinDint[0] := "PLCToEPICS"."Word"[0];
    #MyWordsinDint[1] := "PLCToEPICS"."Word"[1];
    #HashTIAMap := #MyDInt; //Hash from PLCFactory TIA Map


    IF ((#HashIFA = #HashModbus) AND (#HashModbus = #HashTIAMap)) THEN //Check CRCs
        #DEVICE_PARAM_OK := TRUE;
       //##################################### ICS HWI ###############################################
       //############################  ICS Instrument Library     ####################################
       //#  PLC Sample Code in VersionDog: ICS_LIBRARY_MASTER_PLC                                   ##
       //#  CCDB device types: ICS_xxxxx                                                            ##
       //#  EPICS HMI (Block Icons/Faceplates)@ GitLab. Projekt: Cryo / CryogenicsLibrary / CryoLib ##
       //#                                                                                          ##
       //#                                     EH - Alalog Heater                                   ##
       //#                                                                                          ##
       //#                                                                                          ##
       //###########################         Version: 1.3             ################################
       //Author:  Miklos Boros
       //Date:    27-05-2019
       //Version: v1.3
       //Changes:
       //1. Variable name unification
       //###########################         Version: 1.2             ################################
       //Author:  Miklos Boros
       //Date:    28-02-2019
       //Version: v1.2
       //Changes:
       //1. Major review,
       //2. Indent,  unit standardization
       //###########################           Version: 1.1           ################################
       //Author:  Marino Vojneski
       //Date:    2018-07-09
       //Version: v1.1
       //Changes:
       //1. Modified "For OPI visualisation" section: Added digital variable "FB_Keep_Setpoint".
       //2. Modified "Parameter Block" section: Added digital variable "P_Keep_Setpoint".
       //###########################           Version: 1.0           ################################
       //Author:  Miklos Boros, Marino Vojneski
       //Date:    2018-06-12
       //Version: v1.0
       //#############################################################################################
       //###########################
       //STATUS BLOCK
       //###########################
       //Operation modes
       //OPI buttons
       //Setpoint and Manipulated value from HMI

    //********************************************
    //*************STATUS VARIABLES***************
    //********************************************


       #MyWord := W#0;
       #MyBoolsinWord[8] := #"OpMode_Auto";    //EPICSName: OpMode_Auto
       #MyBoolsinWord[9] := #"OpMode_Manual";    //EPICSName: OpMode_Manual
       #MyBoolsinWord[10] := #"OpMode_Forced";    //EPICSName: OpMode_Forced
       "PLCToEPICS"."Word"[#PLCToEPICSDataBlockOffset + 0] := #MyWord;

       #MyReal := #"HeaterCurrent";    //EPICSName: HeaterCurrent
       "PLCToEPICS"."Word"[#PLCToEPICSDataBlockOffset + 1] := #MyWordsinReal[0];
       "PLCToEPICS"."Word"[#PLCToEPICSDataBlockOffset + 2] := #MyWordsinReal[1];

       #MyReal := #"HeaterVoltage";    //EPICSName: HeaterVoltage
       "PLCToEPICS"."Word"[#PLCToEPICSDataBlockOffset + 3] := #MyWordsinReal[0];
       "PLCToEPICS"."Word"[#PLCToEPICSDataBlockOffset + 4] := #MyWordsinReal[1];

       #MyReal := #"HeaterPower";    //EPICSName: HeaterPower
       "PLCToEPICS"."Word"[#PLCToEPICSDataBlockOffset + 5] := #MyWordsinReal[0];
       "PLCToEPICS"."Word"[#PLCToEPICSDataBlockOffset + 6] := #MyWordsinReal[1];

       #MyReal := #"HeaterSP";    //EPICSName: HeaterSP
       "PLCToEPICS"."Word"[#PLCToEPICSDataBlockOffset + 7] := #MyWordsinReal[0];
       "PLCToEPICS"."Word"[#PLCToEPICSDataBlockOffset + 8] := #MyWordsinReal[1];

       #MyReal := #"HeaterMV";    //EPICSName: HeaterMV
       "PLCToEPICS"."Word"[#PLCToEPICSDataBlockOffset + 9] := #MyWordsinReal[0];
       "PLCToEPICS"."Word"[#PLCToEPICSDataBlockOffset + 10] := #MyWordsinReal[1];

       #MyWord := W#0;
       #MyBoolsinWord[8] := #"HeatingON";    //EPICSName: HeatingON
       #MyBoolsinWord[9] := #"Inhibit_Manual";    //EPICSName: Inhibit_Manual
       #MyBoolsinWord[10] := #"Inhibit_Force";    //EPICSName: Inhibit_Force
       #MyBoolsinWord[11] := #"Inhibit_Lock";    //EPICSName: Inhibit_Lock
       #MyBoolsinWord[12] := #"GroupInterlock";    //EPICSName: GroupInterlock
       #MyBoolsinWord[13] := #"HeatInterlock";    //EPICSName: HeatInterlock
       #MyBoolsinWord[14] := #"EnableAutoBtn";    //EPICSName: EnableAutoBtn
       #MyBoolsinWord[15] := #"EnableManualBtn";    //EPICSName: EnableManualBtn
       #MyBoolsinWord[0] := #"EnableForcedBtn";    //EPICSName: EnableForcedBtn
       #MyBoolsinWord[1] := #"EnableForceValBtn";    //EPICSName: EnableForceValBtn
       #MyBoolsinWord[2] := #"DevLocked";    //EPICSName: DevLocked
       "PLCToEPICS"."Word"[#PLCToEPICSDataBlockOffset + 11] := #MyWord;

       #MyDInt := #"Faceplate_LockID";    //EPICSName: Faceplate_LockID
       "PLCToEPICS"."Word"[#PLCToEPICSDataBlockOffset + 12] := #MyWordsinDint[0];
       "PLCToEPICS"."Word"[#PLCToEPICSDataBlockOffset + 13] := #MyWordsinDint[1];

       #MyDInt := #"BlockIcon_LockID";    //EPICSName: BlockIcon_LockID
       "PLCToEPICS"."Word"[#PLCToEPICSDataBlockOffset + 14] := #MyWordsinDint[0];
       "PLCToEPICS"."Word"[#PLCToEPICSDataBlockOffset + 15] := #MyWordsinDint[1];

       #MyWord := W#0;
       #MyBoolsinWord[8] := #"LatchAlarm";    //EPICSName: LatchAlarm
       #MyBoolsinWord[9] := #"GroupAlarm";    //EPICSName: GroupAlarm
       #MyBoolsinWord[10] := #"Power_Discrep";    //EPICSName: Power_Discrep
       #MyBoolsinWord[11] := #"IO_Error";    //EPICSName: IO_Error
       #MyBoolsinWord[12] := #"Input_Module_Error";    //EPICSName: Input_Module_Error
       #MyBoolsinWord[13] := #"Output_Module_Error";    //EPICSName: Output_Module_Error
       "PLCToEPICS"."Word"[#PLCToEPICSDataBlockOffset + 16] := #MyWord;

       #MyReal := #"DiscrPerc";    //EPICSName: DiscrPerc
       "PLCToEPICS"."Word"[#PLCToEPICSDataBlockOffset + 17] := #MyWordsinReal[0];
       "PLCToEPICS"."Word"[#PLCToEPICSDataBlockOffset + 18] := #MyWordsinReal[1];

       #MyTime := #"DiscrTime";    //EPICSName: DiscrTime
       "PLCToEPICS"."Word"[#PLCToEPICSDataBlockOffset + 19] := #MyWordsinTime[0];
       "PLCToEPICS"."Word"[#PLCToEPICSDataBlockOffset + 20] := #MyWordsinTime[1];

       #MyReal := #"MaxRampUPSpd";    //EPICSName: MaxRampUPSpd
       "PLCToEPICS"."Word"[#PLCToEPICSDataBlockOffset + 21] := #MyWordsinReal[0];
       "PLCToEPICS"."Word"[#PLCToEPICSDataBlockOffset + 22] := #MyWordsinReal[1];

       #MyReal := #"MaxRampDNSpd";    //EPICSName: MaxRampDNSpd
       "PLCToEPICS"."Word"[#PLCToEPICSDataBlockOffset + 23] := #MyWordsinReal[0];
       "PLCToEPICS"."Word"[#PLCToEPICSDataBlockOffset + 24] := #MyWordsinReal[1];

       #MyReal := #"ActRampSpeed";    //EPICSName: ActRampSpeed
       "PLCToEPICS"."Word"[#PLCToEPICSDataBlockOffset + 25] := #MyWordsinReal[0];
       "PLCToEPICS"."Word"[#PLCToEPICSDataBlockOffset + 26] := #MyWordsinReal[1];

       #MyWord := W#0;
       #MyBoolsinWord[8] := #"Ramping";    //EPICSName: Ramping
       #MyBoolsinWord[9] := #"RampSettingOK";    //EPICSName: RampSettingOK
       "PLCToEPICS"."Word"[#PLCToEPICSDataBlockOffset + 27] := #MyWord;

       #MyInt := #"FB_RampUPTIME";    //EPICSName: FB_RampUPTIME
       "PLCToEPICS"."Word"[#PLCToEPICSDataBlockOffset + 28] := #MyWordinInt;

       #MyReal := #"FB_RampUPRANGE";    //EPICSName: FB_RampUPRANGE
       "PLCToEPICS"."Word"[#PLCToEPICSDataBlockOffset + 29] := #MyWordsinReal[0];
       "PLCToEPICS"."Word"[#PLCToEPICSDataBlockOffset + 30] := #MyWordsinReal[1];

       #MyInt := #"FB_RampDNTIME";    //EPICSName: FB_RampDNTIME
       "PLCToEPICS"."Word"[#PLCToEPICSDataBlockOffset + 31] := #MyWordinInt;

       #MyReal := #"FB_RampDNRANGE";    //EPICSName: FB_RampDNRANGE
       "PLCToEPICS"."Word"[#PLCToEPICSDataBlockOffset + 32] := #MyWordsinReal[0];
       "PLCToEPICS"."Word"[#PLCToEPICSDataBlockOffset + 33] := #MyWordsinReal[1];

       #MyReal := #"FB_ForcePower";    //EPICSName: FB_ForcePower
       "PLCToEPICS"."Word"[#PLCToEPICSDataBlockOffset + 34] := #MyWordsinReal[0];
       "PLCToEPICS"."Word"[#PLCToEPICSDataBlockOffset + 35] := #MyWordsinReal[1];

       #MyReal := #"FB_Setpoint";    //EPICSName: FB_Setpoint
       "PLCToEPICS"."Word"[#PLCToEPICSDataBlockOffset + 36] := #MyWordsinReal[0];
       "PLCToEPICS"."Word"[#PLCToEPICSDataBlockOffset + 37] := #MyWordsinReal[1];

       #MyReal := #"FB_Manipulated";    //EPICSName: FB_Manipulated
       "PLCToEPICS"."Word"[#PLCToEPICSDataBlockOffset + 38] := #MyWordsinReal[0];
       "PLCToEPICS"."Word"[#PLCToEPICSDataBlockOffset + 39] := #MyWordsinReal[1];

       #MyReal := #"FB_Step";    //EPICSName: FB_Step
       "PLCToEPICS"."Word"[#PLCToEPICSDataBlockOffset + 40] := #MyWordsinReal[0];
       "PLCToEPICS"."Word"[#PLCToEPICSDataBlockOffset + 41] := #MyWordsinReal[1];

       #MyInt := #"FB_RampTIME";    //EPICSName: FB_RampTIME
       "PLCToEPICS"."Word"[#PLCToEPICSDataBlockOffset + 42] := #MyWordinInt;

       #MyReal := #"FB_RampRANGE";    //EPICSName: FB_RampRANGE
       "PLCToEPICS"."Word"[#PLCToEPICSDataBlockOffset + 43] := #MyWordsinReal[0];
       "PLCToEPICS"."Word"[#PLCToEPICSDataBlockOffset + 44] := #MyWordsinReal[1];

    //********************************************
    //*************COMMAND VARIABLES**************
    //********************************************


       #MyWord := "EPICSToPLC"."Word"[#EPICSToPLCDataBlockOffset + 0];
       "EPICSToPLC"."Word"[#EPICSToPLCDataBlockOffset + 0] := 0;
       #"Cmd_Auto" := #MyBoolsinWord[8];    //EPICSName: Cmd_Auto
       #"Cmd_Manual" := #MyBoolsinWord[9];    //EPICSName: Cmd_Manual
       #"Cmd_Force" := #MyBoolsinWord[10];    //EPICSName: Cmd_Force
       #"Cmd_RampON" := #MyBoolsinWord[11];    //EPICSName: Cmd_RampON
       #"Cmd_RampOFF" := #MyBoolsinWord[12];    //EPICSName: Cmd_RampOFF
       #"Cmd_AckAlarm" := #MyBoolsinWord[13];    //EPICSName: Cmd_AckAlarm
       #"Cmd_ForceValInp" := #MyBoolsinWord[14];    //EPICSName: Cmd_ForceValInp
       #"Cmd_ForceValOut" := #MyBoolsinWord[15];    //EPICSName: Cmd_ForceValOut
       #"Cmd_ForceUnlock" := #MyBoolsinWord[0];    //EPICSName: Cmd_ForceUnlock
       #"Cmd_DevLock" := #MyBoolsinWord[1];    //EPICSName: Cmd_DevLock
       #"Cmd_DevUnlock" := #MyBoolsinWord[2];    //EPICSName: Cmd_DevUnlock

    //********************************************
    //************PARAMETER VARIABLES*************
    //********************************************


       #MyReal	:= 0.0;
       #MyWordsinReal[0]	:= "EPICSToPLC"."Word"[#EPICSToPLCDataBlockOffset + 1];
       #MyWordsinReal[1]	:= "EPICSToPLC"."Word"[#EPICSToPLCDataBlockOffset + 2];
       #"P_ForcePower" := #MyReal;    //EPICSName: P_ForcePower

       #MyReal	:= 0.0;
       #MyWordsinReal[0]	:= "EPICSToPLC"."Word"[#EPICSToPLCDataBlockOffset + 3];
       #MyWordsinReal[1]	:= "EPICSToPLC"."Word"[#EPICSToPLCDataBlockOffset + 4];
       #"P_Setpoint" := #MyReal;    //EPICSName: P_Setpoint

       #MyReal	:= 0.0;
       #MyWordsinReal[0]	:= "EPICSToPLC"."Word"[#EPICSToPLCDataBlockOffset + 5];
       #MyWordsinReal[1]	:= "EPICSToPLC"."Word"[#EPICSToPLCDataBlockOffset + 6];
       #"P_Manipulated" := #MyReal;    //EPICSName: P_Manipulated

       #MyReal	:= 0.0;
       #MyWordsinReal[0]	:= "EPICSToPLC"."Word"[#EPICSToPLCDataBlockOffset + 7];
       #MyWordsinReal[1]	:= "EPICSToPLC"."Word"[#EPICSToPLCDataBlockOffset + 8];
       #"P_Step" := #MyReal;    //EPICSName: P_Step

       #MyWordinInt := "EPICSToPLC"."Word"[#EPICSToPLCDataBlockOffset + 9];
       #"P_RampUPTIME" := #MyInt;    //EPICSName: P_RampUPTIME

       #MyReal	:= 0.0;
       #MyWordsinReal[0]	:= "EPICSToPLC"."Word"[#EPICSToPLCDataBlockOffset + 10];
       #MyWordsinReal[1]	:= "EPICSToPLC"."Word"[#EPICSToPLCDataBlockOffset + 11];
       #"P_RampUPRANGE" := #MyReal;    //EPICSName: P_RampUPRANGE

       #MyWordinInt := "EPICSToPLC"."Word"[#EPICSToPLCDataBlockOffset + 12];
       #"P_RampDNTIME" := #MyInt;    //EPICSName: P_RampDNTIME

       #MyReal	:= 0.0;
       #MyWordsinReal[0]	:= "EPICSToPLC"."Word"[#EPICSToPLCDataBlockOffset + 13];
       #MyWordsinReal[1]	:= "EPICSToPLC"."Word"[#EPICSToPLCDataBlockOffset + 14];
       #"P_RampDNRANGE" := #MyReal;    //EPICSName: P_RampDNRANGE

       #MyDInt	:= 0;
       #MyWordsinDint[0]	:= "EPICSToPLC"."Word"[#EPICSToPLCDataBlockOffset + 15];
       #MyWordsinDint[1]	:= "EPICSToPLC"."Word"[#EPICSToPLCDataBlockOffset + 16];
       #"P_Faceplate_LockID" := #MyDInt;    //EPICSName: P_Faceplate_LockID

